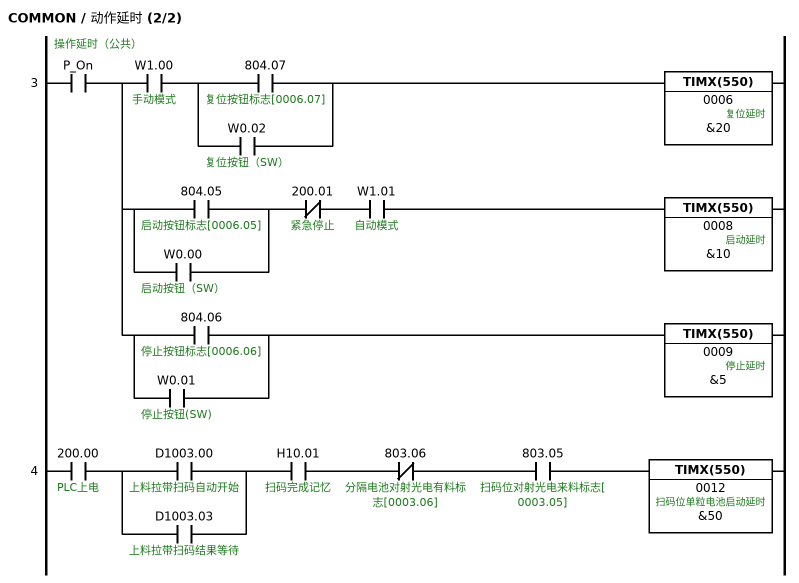
; [picture p168: COMMON / 动作延时, rungs 3-4]
; rung 3: 操作延时（公共）
LD P_On
OUT TR0
AND W1.00  ; 手动模式
LD 804.07  ; 复位按钮标志[0006.07]
OR W0.02  ; 复位按钮（SW）
ANDLD
TIMX(550) 0006 &20  ; 复位延时
LD TR0
LD 804.05  ; 启动按钮标志[0006.05]
OR W0.00  ; 启动按钮（SW）
ANDLD
ANDNOT 200.01  ; 紧急停止
AND W1.01  ; 自动模式
TIMX(550) 0008 &10  ; 启动延时
LD TR0
LD 804.06  ; 停止按钮标志[0006.06]
OR W0.01  ; 停止按钮(SW)
ANDLD
TIMX(550) 0009 &5  ; 停止延时
; rung 4
LD 200.00  ; PLC上电
LD D1003.00  ; 上料拉带扫码自动开始
OR D1003.03  ; 上料拉带扫码结果等待
ANDLD
AND H10.01  ; 扫码完成记忆
ANDNOT 803.06  ; 分隔电池对射光电有料标志[0003.06]
AND 803.05  ; 扫码位对射光电来料标志[0003.05]
TIMX(550) 0012 &50  ; 扫码位单粒电池启动延时

### Section 数据传输

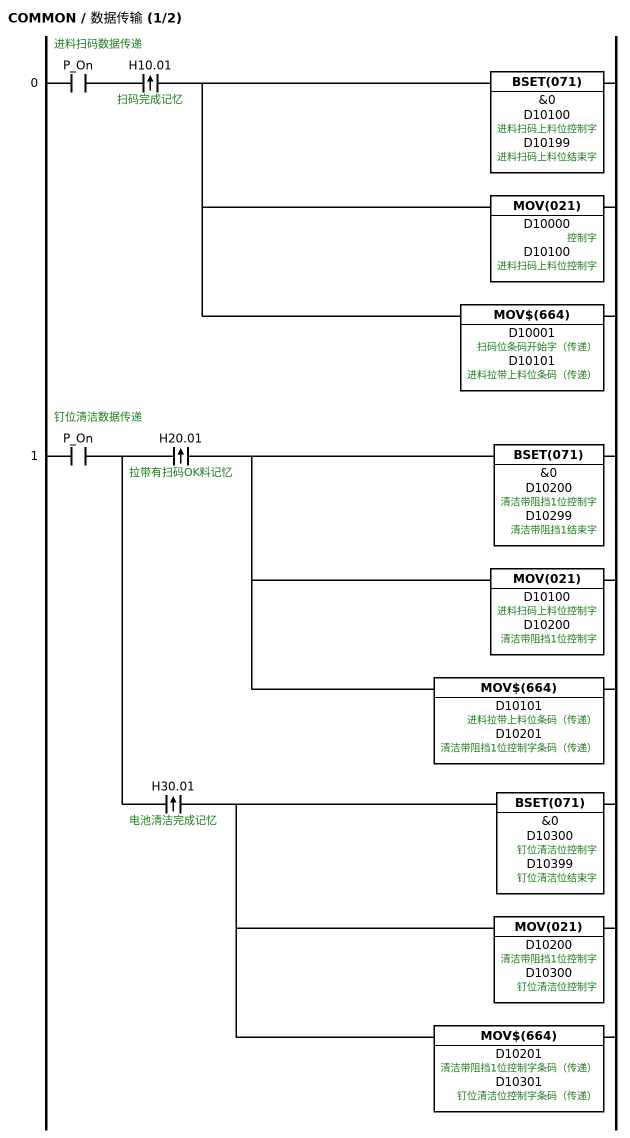
; rung 0: 进料扫码数据传递
LD P_On
@AND H10.01  ; 扫码完成记忆
BSET(071) &0 D10100 D10199  ; 进料扫码上料位控制字, 进料扫码上料位结束字
MOV(021) D10000 D10100  ; 控制字, 进料扫码上料位控制字
MOV$(664) D10001 D10101  ; 扫码位条码开始字（传递）, 进料拉带上料位条码（传递）
; rung 1: 钉位清洁数据传递
LD P_On
OUT TR0
@AND H20.01  ; 拉带有扫码OK料记忆
BSET(071) &0 D10200 D10299  ; 清洁带阻挡1位控制字, 清洁带阻挡1结束字
MOV(021) D10100 D10200  ; 进料扫码上料位控制字, 清洁带阻挡1位控制字
MOV$(664) D10101 D10201  ; 进料拉带上料位条码（传递）, 清洁带阻挡1位控制字条码（传递）
LD TR0
@AND H30.01  ; 电池清洁完成记忆
BSET(071) &0 D10300 D10399  ; 钉位清洁位控制字, 钉位清洁位结束字
MOV(021) D10200 D10300  ; 清洁带阻挡1位控制字, 钉位清洁位控制字
MOV$(664) D10201 D10301  ; 清洁带阻挡1位控制字条码（传递）, 钉位清洁位控制字条码（传递）

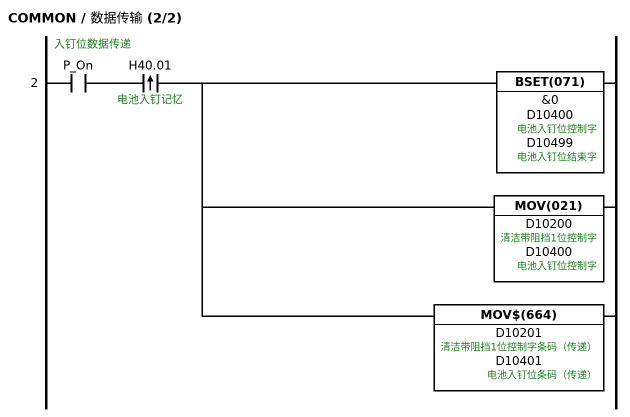
; rung 2: 入钉位数据传递
LD P_On
@AND H40.01  ; 电池入钉记忆
BSET(071) &0 D10400 D10499  ; 电池入钉位控制字, 电池入钉位结束字
MOV(021) D10200 D10400  ; 清洁带阻挡1位控制字, 电池入钉位控制字
MOV$(664) D10201 D10401  ; 清洁带阻挡1位控制字条码（传递）, 电池入钉位条码（传递）

### Section 数据处理

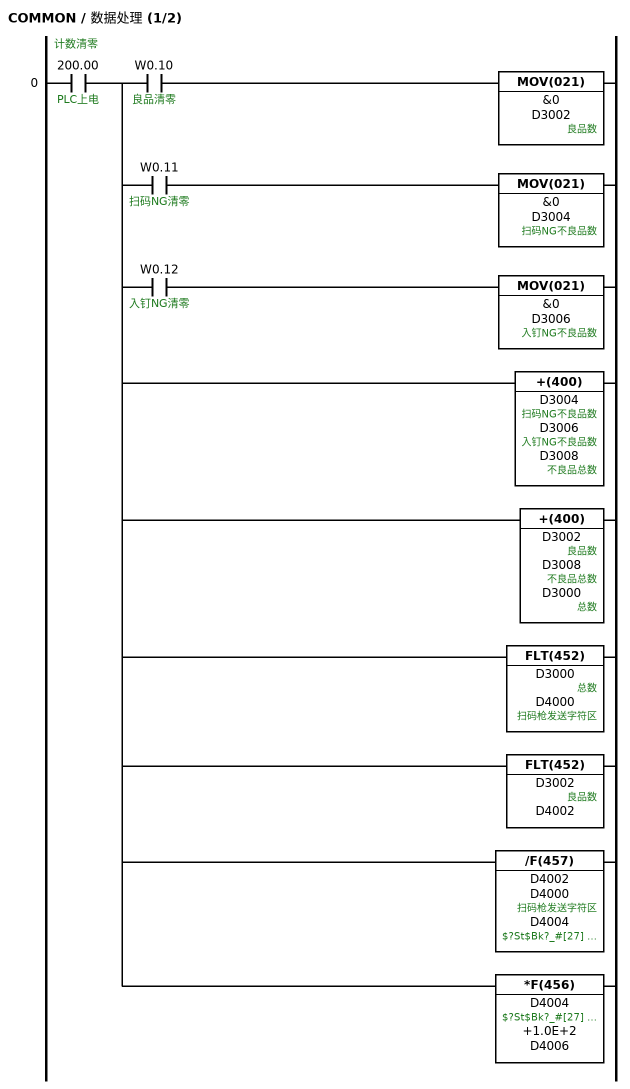
; rung 0: 计数清零
LD 200.00  ; PLC上电
OUT TR0
AND W0.10  ; 良品清零
MOV(021) &0 D3002  ; 良品数
LD TR0
AND W0.11  ; 扫码NG清零
MOV(021) &0 D3004  ; 扫码NG不良品数
LD TR0
AND W0.12  ; 入钉NG清零
MOV(021) &0 D3006  ; 入钉NG不良品数
LD TR0
+(400) D3004 D3006 D3008  ; 扫码NG不良品数, 入钉NG不良品数, 不良品总数
+(400) D3002 D3008 D3000  ; 良品数, 不良品总数, 总数
FLT(452) D3000 D4000  ; 总数, 扫码枪发送字符区
FLT(452) D3002 D4002  ; 良品数
/F(457) D4002 D4000 D4004  ; 扫码枪发送字符区, $?St$Bk?_#[27] / "OK"$?St$Bk?_#[27]
*F(456) D4004 +1.0E+2 D4006  ; $?St$Bk?_#[27] / "OK"$?St$Bk?_#[27]

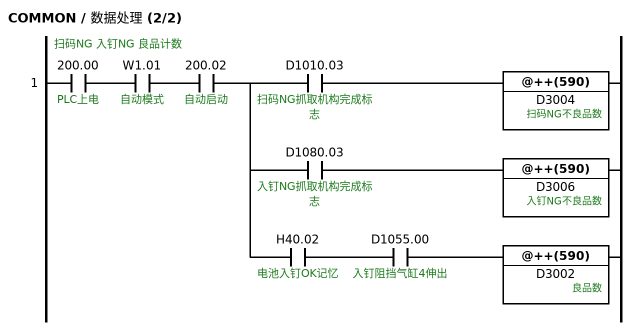
; rung 1: 扫码NG 入钉NG 良品计数
LD 200.00  ; PLC上电
AND W1.01  ; 自动模式
AND 200.02  ; 自动启动
OUT TR0
AND D1010.03  ; 扫码NG抓取机构完成标志
@++(590) D3004  ; 扫码NG不良品数
LD TR0
AND D1080.03  ; 入钉NG抓取机构完成标志
@++(590) D3006  ; 入钉NG不良品数
LD TR0
AND H40.02  ; 电池入钉OK记忆
AND D1055.00  ; 入钉阻挡气缸4伸出
@++(590) D3002  ; 良品数

### Section 报警程序

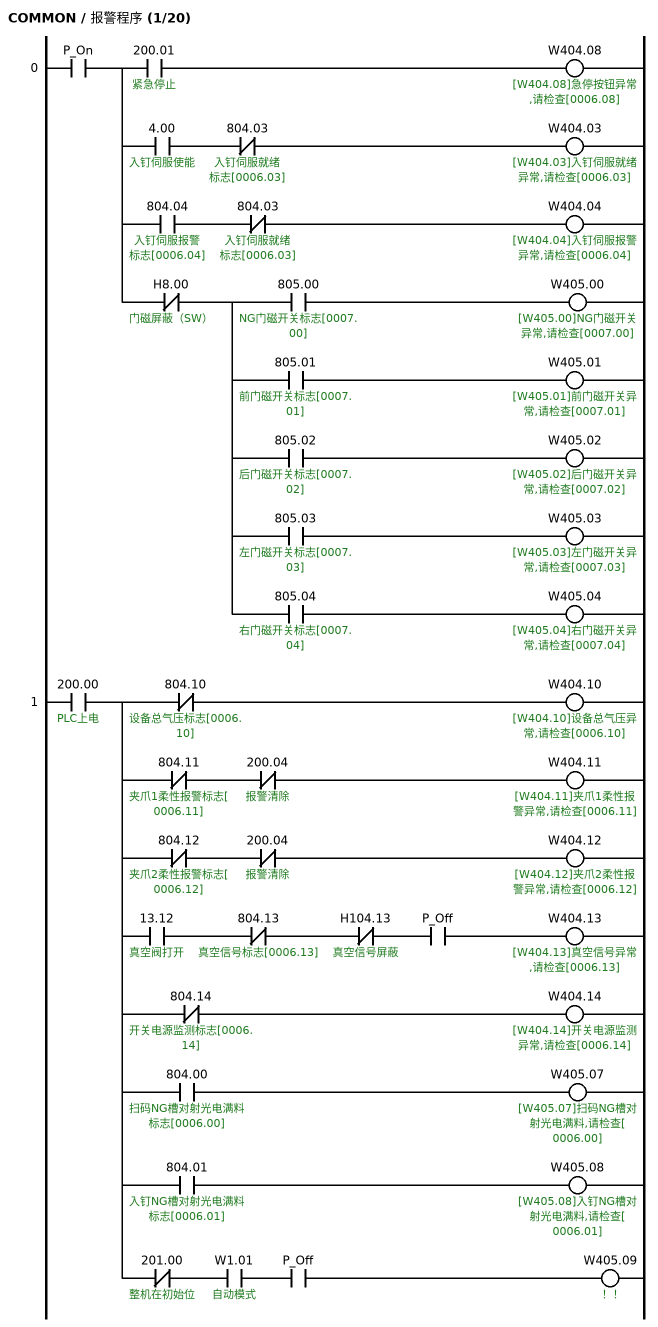
; rung 0
LD P_On
OUT TR0
AND 200.01  ; 紧急停止
OUT W404.08  ; [W404.08]急停按钮异常,请检查[0006.08]
LD TR0
AND 4.00  ; 入钉伺服使能
ANDNOT 804.03  ; 入钉伺服就绪 标志[0006.03]
OUT W404.03  ; [W404.03]入钉伺服就绪异常,请检查[0006.03]
LD TR0
AND 804.04  ; 入钉伺服报警 标志[0006.04]
ANDNOT 804.03  ; 入钉伺服就绪 标志[0006.03]
OUT W404.04  ; [W404.04]入钉伺服报警异常,请检查[0006.04]
LD TR0
ANDNOT H8.00  ; 门磁屏蔽（SW）
OUT TR0
AND 805.00  ; NG门磁开关标志[0007.00]
OUT W405.00  ; [W405.00]NG门磁开关异常,请检查[0007.00]
LD TR0
AND 805.01  ; 前门磁开关标志[0007.01]
OUT W405.01  ; [W405.01]前门磁开关异常,请检查[0007.01]
LD TR0
AND 805.02  ; 后门磁开关标志[0007.02]
OUT W405.02  ; [W405.02]后门磁开关异常,请检查[0007.02]
LD TR0
AND 805.03  ; 左门磁开关标志[0007.03]
OUT W405.03  ; [W405.03]左门磁开关异常,请检查[0007.03]
LD TR0
AND 805.04  ; 右门磁开关标志[0007.04]
OUT W405.04  ; [W405.04]右门磁开关异常,请检查[0007.04]
; rung 1
LD 200.00  ; PLC上电
OUT TR0
ANDNOT 804.10  ; 设备总气压标志[0006.10]
OUT W404.10  ; [W404.10]设备总气压异常,请检查[0006.10]
LD TR0
ANDNOT 804.11  ; 夹爪1柔性报警标志[0006.11]
ANDNOT 200.04  ; 报警清除
OUT W404.11  ; [W404.11]夹爪1柔性报警异常,请检查[0006.11]
LD TR0
ANDNOT 804.12  ; 夹爪2柔性报警标志[0006.12]
ANDNOT 200.04  ; 报警清除
OUT W404.12  ; [W404.12]夹爪2柔性报警异常,请检查[0006.12]
LD TR0
AND 13.12  ; 真空阀打开
ANDNOT 804.13  ; 真空信号标志[0006.13]
ANDNOT H104.13  ; 真空信号屏蔽
AND P_Off
OUT W404.13  ; [W404.13]真空信号异常,请检查[0006.13]
LD TR0
ANDNOT 804.14  ; 开关电源监测标志[0006.14]
OUT W404.14  ; [W404.14]开关电源监测异常,请检查[0006.14]
LD TR0
AND 804.00  ; 扫码NG槽对射光电满料标志[0006.00]
OUT W405.07  ; [W405.07]扫码NG槽对射光电满料,请检查[0006.00]
LD TR0
AND 804.01  ; 入钉NG槽对射光电满料标志[0006.01]
OUT W405.08  ; [W405.08]入钉NG槽对射光电满料,请检查[0006.01]
LD TR0
ANDNOT 201.00  ; 整机在初始位
AND W1.01  ; 自动模式
AND P_Off
OUT W405.09  ; ！！

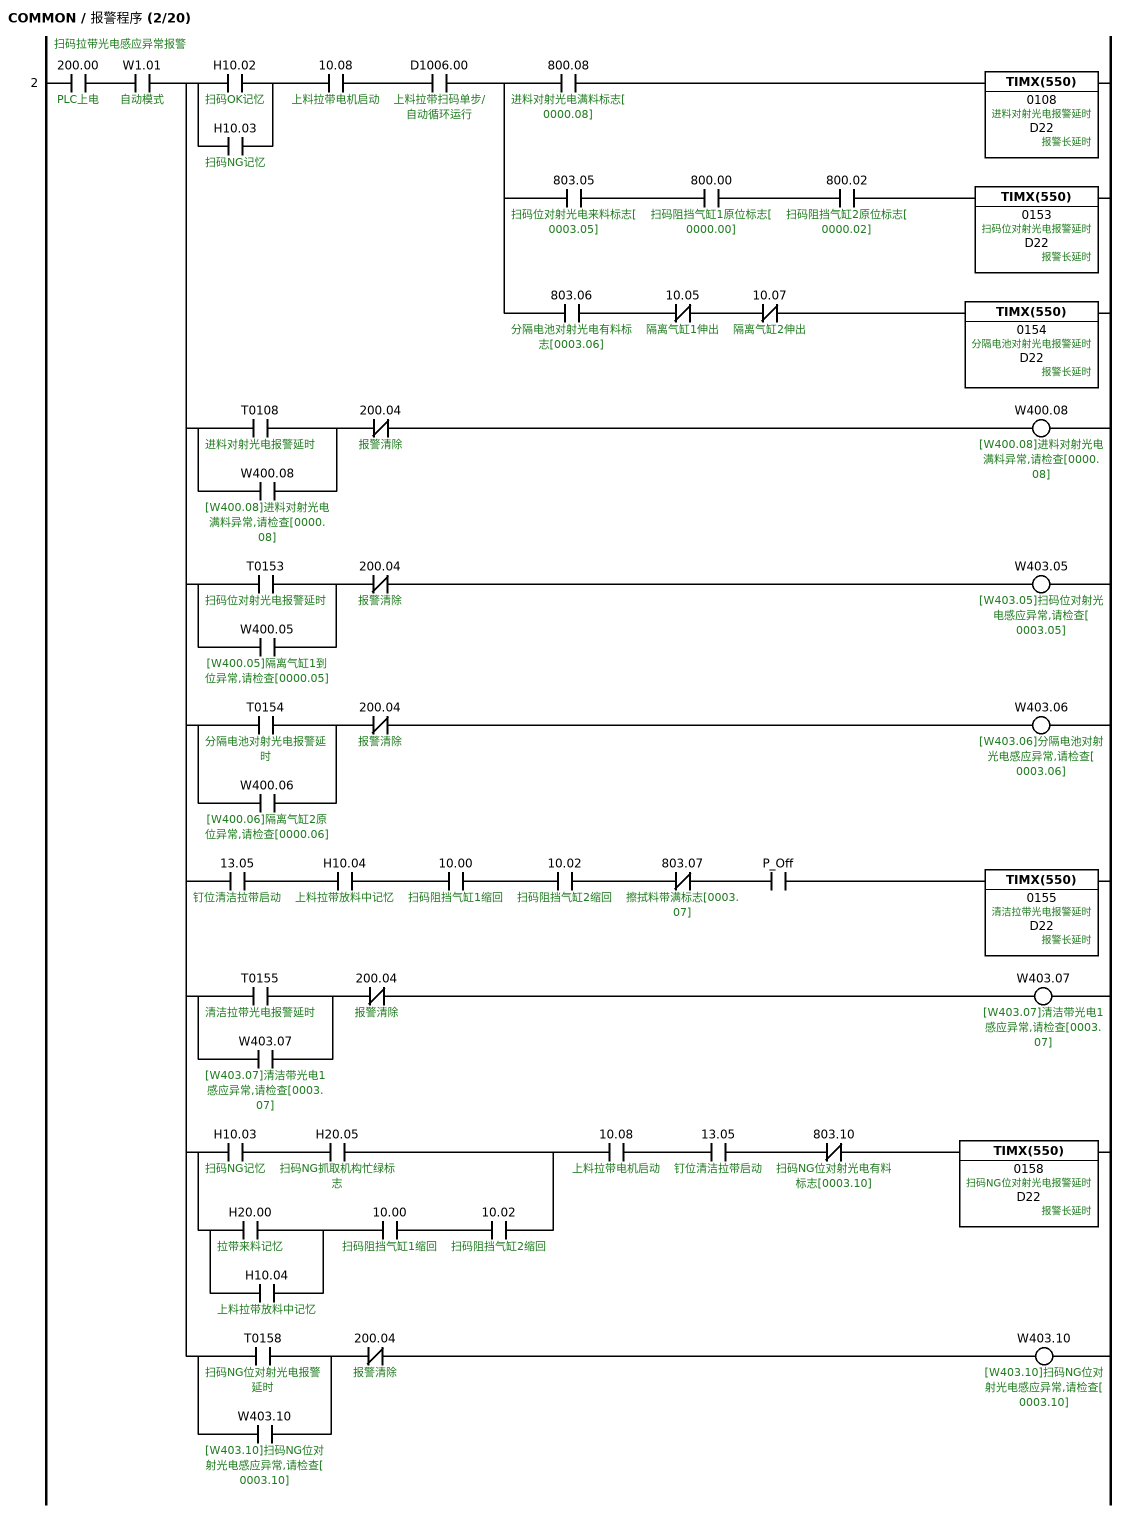
; rung 2: 扫码拉带光电感应异常报警
LD 200.00  ; PLC上电
AND W1.01  ; 自动模式
OUT TR0
LD H10.02  ; 扫码OK记忆
OR H10.03  ; 扫码NG记忆
ANDLD
AND 10.08  ; 上料拉带电机启动
AND D1006.00  ; 上料拉带扫码单步/自动循环运行
OUT TR1
AND 800.08  ; 进料对射光电满料标志[0000.08]
TIMX(550) 0108 D22  ; 报警长延时, 进料对射光电报警延时
LD TR1
AND 803.05  ; 扫码位对射光电来料标志[0003.05]
AND 800.00  ; 扫码阻挡气缸1原位标志[0000.00]
AND 800.02  ; 扫码阻挡气缸2原位标志[0000.02]
TIMX(550) 0153 D22  ; 报警长延时, 扫码位对射光电报警延时
LD TR1
AND 803.06  ; 分隔电池对射光电有料标志[0003.06]
ANDNOT 10.05  ; 隔离气缸1伸出
ANDNOT 10.07  ; 隔离气缸2伸出
TIMX(550) 0154 D22  ; 报警长延时, 分隔电池对射光电报警延时
LD TR0
LD T0108  ; 进料对射光电报警延时
OR W400.08  ; [W400.08]进料对射光电满料异常,请检查[0000.08]
ANDLD
ANDNOT 200.04  ; 报警清除
OUT W400.08  ; [W400.08]进料对射光电满料异常,请检查[0000.08]
LD TR0
LD T0153  ; 扫码位对射光电报警延时
OR W400.05  ; [W400.05]隔离气缸1到位异常,请检查[0000.05]
ANDLD
ANDNOT 200.04  ; 报警清除
OUT W403.05  ; [W403.05]扫码位对射光电感应异常,请检查[0003.05]
LD TR0
LD T0154  ; 分隔电池对射光电报警延时
OR W400.06  ; [W400.06]隔离气缸2原位异常,请检查[0000.06]
ANDLD
ANDNOT 200.04  ; 报警清除
OUT W403.06  ; [W403.06]分隔电池对射光电感应异常,请检查[0003.06]
LD TR0
AND 13.05  ; 钉位清洁拉带启动
AND H10.04  ; 上料拉带放料中记忆
AND 10.00  ; 扫码阻挡气缸1缩回
AND 10.02  ; 扫码阻挡气缸2缩回
ANDNOT 803.07  ; 擦拭料带满标志[0003.07]
AND P_Off
TIMX(550) 0155 D22  ; 报警长延时, 清洁拉带光电报警延时
LD TR0
LD T0155  ; 清洁拉带光电报警延时
OR W403.07  ; [W403.07]清洁带光电1感应异常,请检查[0003.07]
ANDLD
ANDNOT 200.04  ; 报警清除
OUT W403.07  ; [W403.07]清洁带光电1感应异常,请检查[0003.07]
LD TR0
LD H10.03  ; 扫码NG记忆
AND H20.05  ; 扫码NG抓取机构忙绿标志
LD H20.00  ; 拉带来料记忆
OR H10.04  ; 上料拉带放料中记忆
AND 10.00  ; 扫码阻挡气缸1缩回
AND 10.02  ; 扫码阻挡气缸2缩回
ORLD
ANDLD
AND 10.08  ; 上料拉带电机启动
AND 13.05  ; 钉位清洁拉带启动
ANDNOT 803.10  ; 扫码NG位对射光电有料标志[0003.10]
TIMX(550) 0158 D22  ; 报警长延时, 扫码NG位对射光电报警延时
LD TR0
LD T0158  ; 扫码NG位对射光电报警延时
OR W403.10  ; [W403.10]扫码NG位对射光电感应异常,请检查[0003.10]
ANDLD
ANDNOT 200.04  ; 报警清除
OUT W403.10  ; [W403.10]扫码NG位对射光电感应异常,请检查[0003.10]

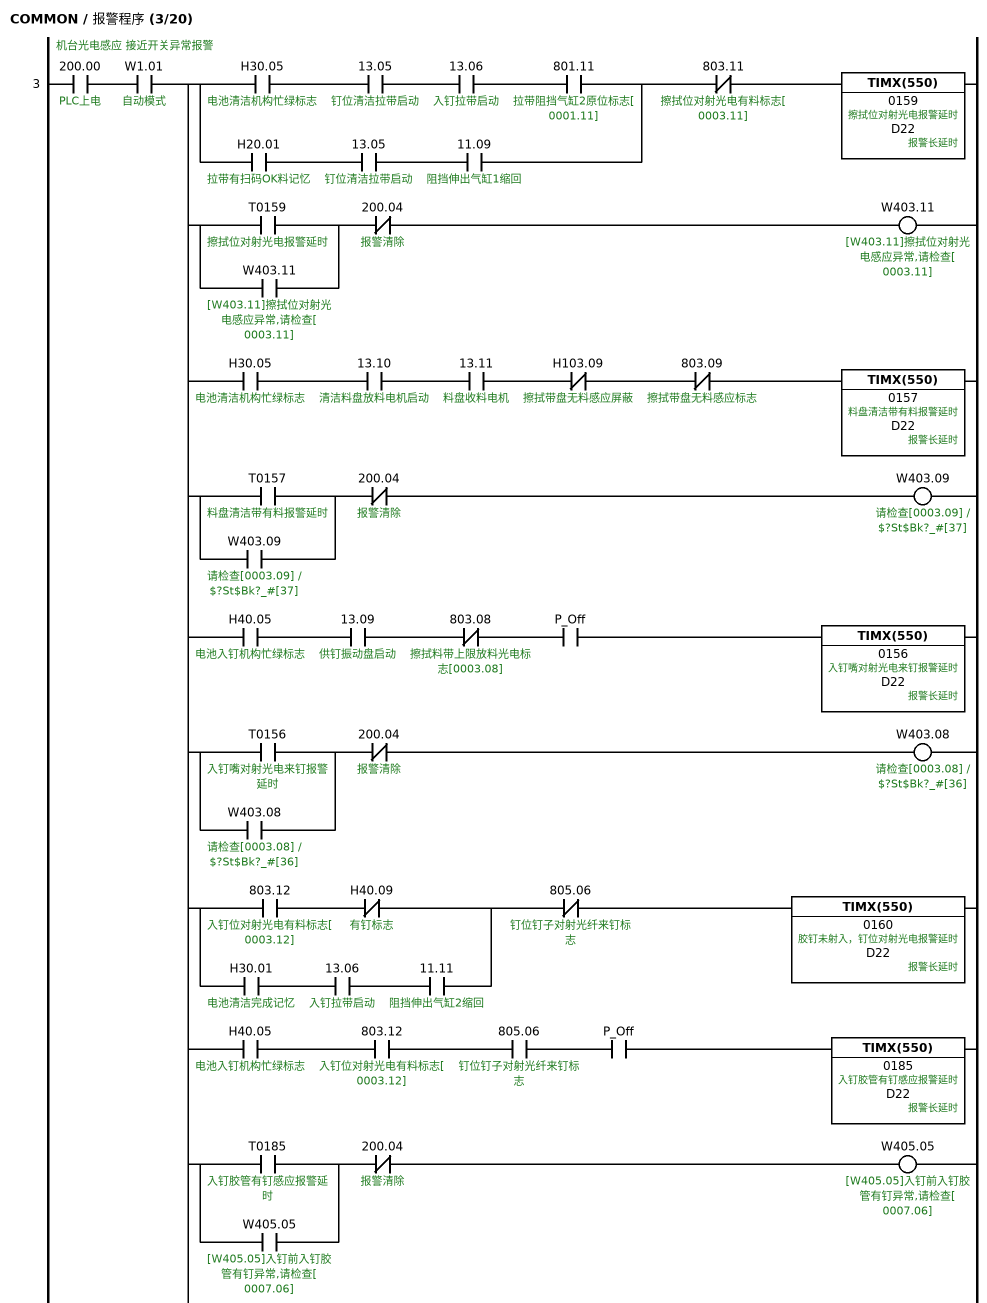

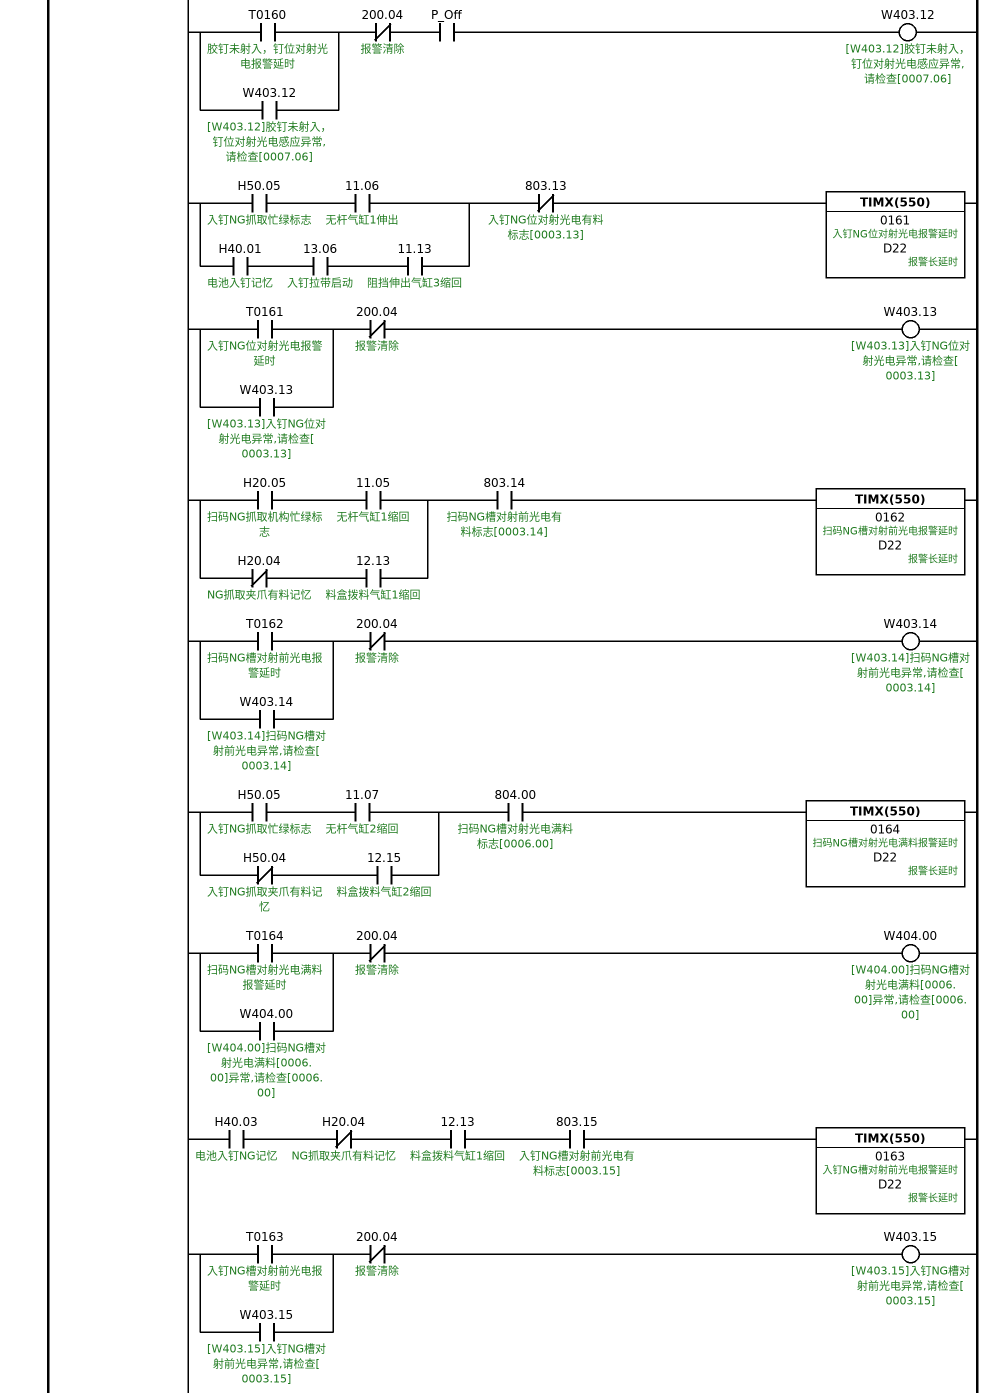

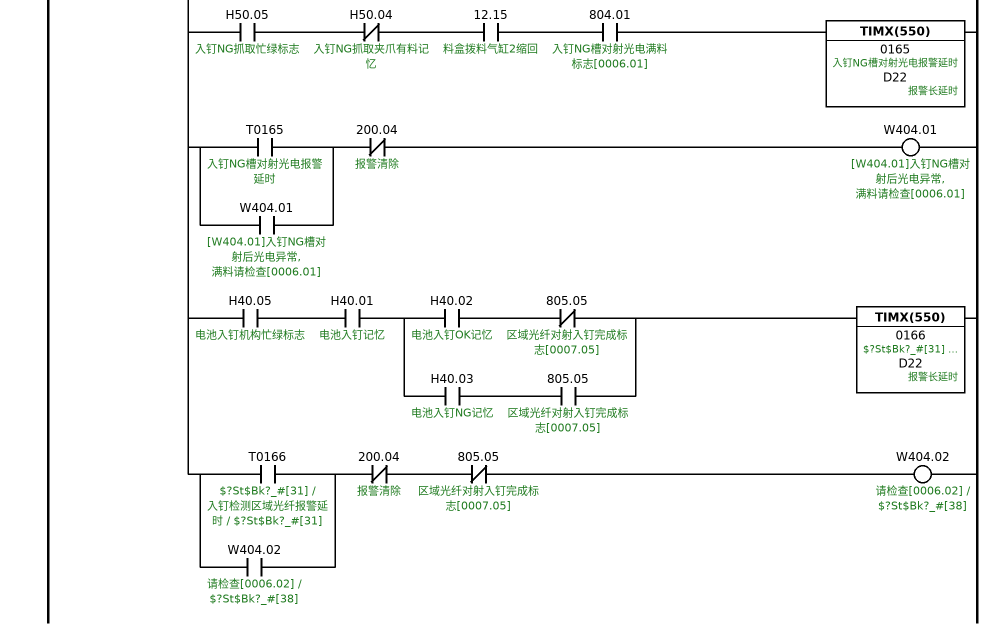
; rung 3: 机台光电感应 接近开关异常报警
LD 200.00  ; PLC上电
AND W1.01  ; 自动模式
OUT TR0
LD H30.05  ; 电池清洁机构忙绿标志
AND 13.05  ; 钉位清洁拉带启动
AND 13.06  ; 入钉拉带启动
AND 801.11  ; 拉带阻挡气缸2原位标志[0001.11]
LD H20.01  ; 拉带有扫码OK料记忆
AND 13.05  ; 钉位清洁拉带启动
AND 11.09  ; 阻挡伸出气缸1缩回
ORLD
ANDLD
ANDNOT 803.11  ; 擦拭位对射光电有料标志[0003.11]
TIMX(550) 0159 D22  ; 报警长延时, 擦拭位对射光电报警延时
LD TR0
LD T0159  ; 擦拭位对射光电报警延时
OR W403.11  ; [W403.11]擦拭位对射光电感应异常,请检查[0003.11]
ANDLD
ANDNOT 200.04  ; 报警清除
OUT W403.11  ; [W403.11]擦拭位对射光电感应异常,请检查[0003.11]
LD TR0
AND H30.05  ; 电池清洁机构忙绿标志
AND 13.10  ; 清洁料盘放料电机启动
AND 13.11  ; 料盘收料电机
ANDNOT H103.09  ; 擦拭带盘无料感应屏蔽
ANDNOT 803.09  ; 擦拭带盘无料感应标志
TIMX(550) 0157 D22  ; 报警长延时, 料盘清洁带有料报警延时
LD TR0
LD T0157  ; 料盘清洁带有料报警延时
OR W403.09  ; 请检查[0003.09] / $?St$Bk?_#[37]
ANDLD
ANDNOT 200.04  ; 报警清除
OUT W403.09  ; 请检查[0003.09] / $?St$Bk?_#[37]
LD TR0
AND H40.05  ; 电池入钉机构忙绿标志
AND 13.09  ; 供钉振动盘启动
ANDNOT 803.08  ; 擦拭料带上限放料光电标志[0003.08]
AND P_Off
TIMX(550) 0156 D22  ; 报警长延时, 入钉嘴对射光电来钉报警延时
LD TR0
LD T0156  ; 入钉嘴对射光电来钉报警延时
OR W403.08  ; 请检查[0003.08] / $?St$Bk?_#[36]
ANDLD
ANDNOT 200.04  ; 报警清除
OUT W403.08  ; 请检查[0003.08] / $?St$Bk?_#[36]
LD TR0
LD 803.12  ; 入钉位对射光电有料标志[0003.12]
ANDNOT H40.09  ; 有钉标志
LD H30.01  ; 电池清洁完成记忆
AND 13.06  ; 入钉拉带启动
AND 11.11  ; 阻挡伸出气缸2缩回
ORLD
ANDLD
ANDNOT 805.06  ; 钉位钉子对射光纤来钉标志
TIMX(550) 0160 D22  ; 报警长延时, 胶钉未射入，钉位对射光电报警延时
LD TR0
AND H40.05  ; 电池入钉机构忙绿标志
AND 803.12  ; 入钉位对射光电有料标志[0003.12]
AND 805.06  ; 钉位钉子对射光纤来钉标志
AND P_Off
TIMX(550) 0185 D22  ; 报警长延时, 入钉胶管有钉感应报警延时
LD TR0
LD T0185  ; 入钉胶管有钉感应报警延时
OR W405.05  ; [W405.05]入钉前入钉胶管有钉异常,请检查[0007.06]
ANDLD
ANDNOT 200.04  ; 报警清除
OUT W405.05  ; [W405.05]入钉前入钉胶管有钉异常,请检查[0007.06]
LD TR0
LD T0160  ; 胶钉未射入，钉位对射光电报警延时
OR W403.12  ; [W403.12]胶钉未射入，钉位对射光电感应异常,请检查[0007.06]
ANDLD
ANDNOT 200.04  ; 报警清除
AND P_Off
OUT W403.12  ; [W403.12]胶钉未射入，钉位对射光电感应异常,请检查[0007.06]
LD TR0
LD H50.05  ; 入钉NG抓取忙绿标志
AND 11.06  ; 无杆气缸1伸出
LD H40.01  ; 电池入钉记忆
AND 13.06  ; 入钉拉带启动
AND 11.13  ; 阻挡伸出气缸3缩回
ORLD
ANDLD
ANDNOT 803.13  ; 入钉NG位对射光电有料标志[0003.13]
TIMX(550) 0161 D22  ; 报警长延时, 入钉NG位对射光电报警延时
LD TR0
LD T0161  ; 入钉NG位对射光电报警延时
OR W403.13  ; [W403.13]入钉NG位对射光电异常,请检查[0003.13]
ANDLD
ANDNOT 200.04  ; 报警清除
OUT W403.13  ; [W403.13]入钉NG位对射光电异常,请检查[0003.13]
LD TR0
LD H20.05  ; 扫码NG抓取机构忙绿标志
AND 11.05  ; 无杆气缸1缩回
LDNOT H20.04  ; NG抓取夹爪有料记忆
AND 12.13  ; 料盒拨料气缸1缩回
ORLD
ANDLD
AND 803.14  ; 扫码NG槽对射前光电有料标志[0003.14]
TIMX(550) 0162 D22  ; 报警长延时, 扫码NG槽对射前光电报警延时
LD TR0
LD T0162  ; 扫码NG槽对射前光电报警延时
OR W403.14  ; [W403.14]扫码NG槽对射前光电异常,请检查[0003.14]
ANDLD
ANDNOT 200.04  ; 报警清除
OUT W403.14  ; [W403.14]扫码NG槽对射前光电异常,请检查[0003.14]
LD TR0
LD H50.05  ; 入钉NG抓取忙绿标志
AND 11.07  ; 无杆气缸2缩回
LDNOT H50.04  ; 入钉NG抓取夹爪有料记忆
AND 12.15  ; 料盒拨料气缸2缩回
ORLD
ANDLD
AND 804.00  ; 扫码NG槽对射光电满料标志[0006.00]
TIMX(550) 0164 D22  ; 报警长延时, 扫码NG槽对射光电满料报警延时
LD TR0
LD T0164  ; 扫码NG槽对射光电满料报警延时
OR W404.00  ; [W404.00]扫码NG槽对射光电满料[0006.00]异常,请检查[0006.00]
ANDLD
ANDNOT 200.04  ; 报警清除
OUT W404.00  ; [W404.00]扫码NG槽对射光电满料[0006.00]异常,请检查[0006.00]
LD TR0
AND H40.03  ; 电池入钉NG记忆
ANDNOT H20.04  ; NG抓取夹爪有料记忆
AND 12.13  ; 料盒拨料气缸1缩回
AND 803.15  ; 入钉NG槽对射前光电有料标志[0003.15]
TIMX(550) 0163 D22  ; 报警长延时, 入钉NG槽对射前光电报警延时
LD TR0
LD T0163  ; 入钉NG槽对射前光电报警延时
OR W403.15  ; [W403.15]入钉NG槽对射前光电异常,请检查[0003.15]
ANDLD
ANDNOT 200.04  ; 报警清除
OUT W403.15  ; [W403.15]入钉NG槽对射前光电异常,请检查[0003.15]
LD TR0
AND H50.05  ; 入钉NG抓取忙绿标志
ANDNOT H50.04  ; 入钉NG抓取夹爪有料记忆
AND 12.15  ; 料盒拨料气缸2缩回
AND 804.01  ; 入钉NG槽对射光电满料标志[0006.01]
TIMX(550) 0165 D22  ; 报警长延时, 入钉NG槽对射光电报警延时
LD TR0
LD T0165  ; 入钉NG槽对射光电报警延时
OR W404.01  ; [W404.01]入钉NG槽对射后光电异常,满料请检查[0006.01]
ANDLD
ANDNOT 200.04  ; 报警清除
OUT W404.01  ; [W404.01]入钉NG槽对射后光电异常,满料请检查[0006.01]
LD TR0
AND H40.05  ; 电池入钉机构忙绿标志
AND H40.01  ; 电池入钉记忆
LD H40.02  ; 电池入钉OK记忆
ANDNOT 805.05  ; 区域光纤对射入钉完成标志[0007.05]
LD H40.03  ; 电池入钉NG记忆
AND 805.05  ; 区域光纤对射入钉完成标志[0007.05]
ORLD
ANDLD
TIMX(550) 0166 D22  ; 报警长延时, $?St$Bk?_#[31] / 入钉检测区域光纤报警延时 / $?St$Bk?_#[31]
LD TR0
LD T0166  ; $?St$Bk?_#[31] / 入钉检测区域光纤报警延时 / $?St$Bk?_#[31]
OR W404.02  ; 请检查[0006.02] / $?St$Bk?_#[38]
ANDLD
ANDNOT 200.04  ; 报警清除
ANDNOT 805.05  ; 区域光纤对射入钉完成标志[0007.05]
OUT W404.02  ; 请检查[0006.02] / $?St$Bk?_#[38]

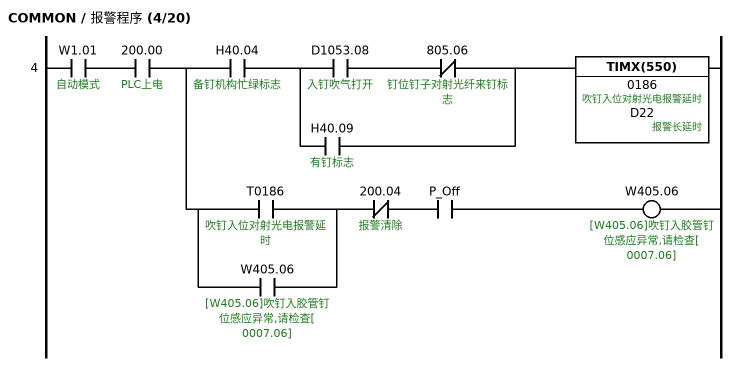
; rung 4
LD W1.01  ; 自动模式
AND 200.00  ; PLC上电
OUT TR0
AND H40.04  ; 备钉机构忙绿标志
LD D1053.08  ; 入钉吹气打开
ANDNOT 805.06  ; 钉位钉子对射光纤来钉标志
OR H40.09  ; 有钉标志
ANDLD
TIMX(550) 0186 D22  ; 报警长延时, 吹钉入位对射光电报警延时
LD TR0
LD T0186  ; 吹钉入位对射光电报警延时
OR W405.06  ; [W405.06]吹钉入胶管钉位感应异常,请检查[0007.06]
ANDLD
ANDNOT 200.04  ; 报警清除
AND P_Off
OUT W405.06  ; [W405.06]吹钉入胶管钉位感应异常,请检查[0007.06]

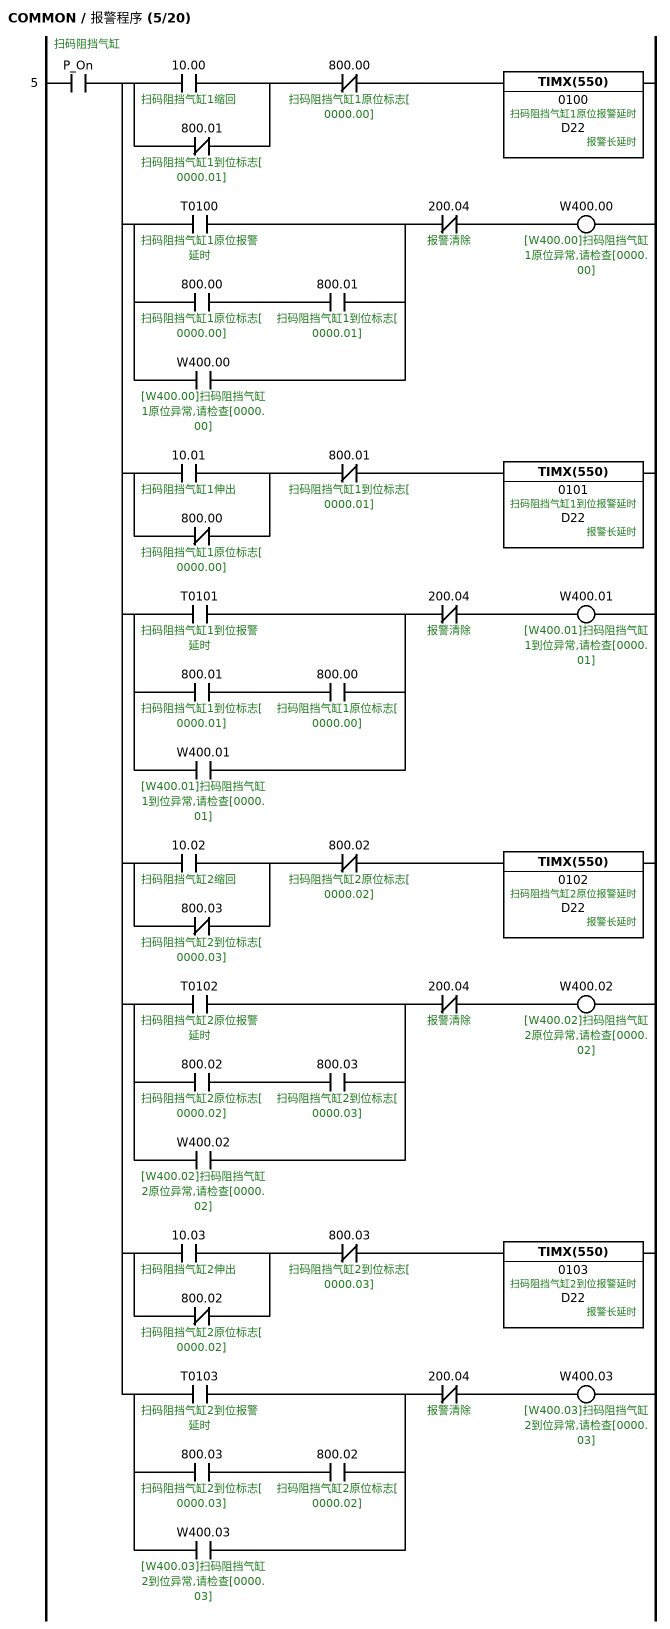
; rung 5: 扫码阻挡气缸
LD P_On
OUT TR0
LD 10.00  ; 扫码阻挡气缸1缩回
ORNOT 800.01  ; 扫码阻挡气缸1到位标志[0000.01]
ANDLD
ANDNOT 800.00  ; 扫码阻挡气缸1原位标志[0000.00]
TIMX(550) 0100 D22  ; 报警长延时, 扫码阻挡气缸1原位报警延时
LD TR0
LD T0100  ; 扫码阻挡气缸1原位报警延时
LD 800.00  ; 扫码阻挡气缸1原位标志[0000.00]
AND 800.01  ; 扫码阻挡气缸1到位标志[0000.01]
ORLD
OR W400.00  ; [W400.00]扫码阻挡气缸1原位异常,请检查[0000.00]
ANDLD
ANDNOT 200.04  ; 报警清除
OUT W400.00  ; [W400.00]扫码阻挡气缸1原位异常,请检查[0000.00]
LD TR0
LD 10.01  ; 扫码阻挡气缸1伸出
ORNOT 800.00  ; 扫码阻挡气缸1原位标志[0000.00]
ANDLD
ANDNOT 800.01  ; 扫码阻挡气缸1到位标志[0000.01]
TIMX(550) 0101 D22  ; 报警长延时, 扫码阻挡气缸1到位报警延时
LD TR0
LD T0101  ; 扫码阻挡气缸1到位报警延时
LD 800.01  ; 扫码阻挡气缸1到位标志[0000.01]
AND 800.00  ; 扫码阻挡气缸1原位标志[0000.00]
ORLD
OR W400.01  ; [W400.01]扫码阻挡气缸1到位异常,请检查[0000.01]
ANDLD
ANDNOT 200.04  ; 报警清除
OUT W400.01  ; [W400.01]扫码阻挡气缸1到位异常,请检查[0000.01]
LD TR0
LD 10.02  ; 扫码阻挡气缸2缩回
ORNOT 800.03  ; 扫码阻挡气缸2到位标志[0000.03]
ANDLD
ANDNOT 800.02  ; 扫码阻挡气缸2原位标志[0000.02]
TIMX(550) 0102 D22  ; 报警长延时, 扫码阻挡气缸2原位报警延时
LD TR0
LD T0102  ; 扫码阻挡气缸2原位报警延时
LD 800.02  ; 扫码阻挡气缸2原位标志[0000.02]
AND 800.03  ; 扫码阻挡气缸2到位标志[0000.03]
ORLD
OR W400.02  ; [W400.02]扫码阻挡气缸2原位异常,请检查[0000.02]
ANDLD
ANDNOT 200.04  ; 报警清除
OUT W400.02  ; [W400.02]扫码阻挡气缸2原位异常,请检查[0000.02]
LD TR0
LD 10.03  ; 扫码阻挡气缸2伸出
ORNOT 800.02  ; 扫码阻挡气缸2原位标志[0000.02]
ANDLD
ANDNOT 800.03  ; 扫码阻挡气缸2到位标志[0000.03]
TIMX(550) 0103 D22  ; 报警长延时, 扫码阻挡气缸2到位报警延时
LD TR0
LD T0103  ; 扫码阻挡气缸2到位报警延时
LD 800.03  ; 扫码阻挡气缸2到位标志[0000.03]
AND 800.02  ; 扫码阻挡气缸2原位标志[0000.02]
ORLD
OR W400.03  ; [W400.03]扫码阻挡气缸2到位异常,请检查[0000.03]
ANDLD
ANDNOT 200.04  ; 报警清除
OUT W400.03  ; [W400.03]扫码阻挡气缸2到位异常,请检查[0000.03]

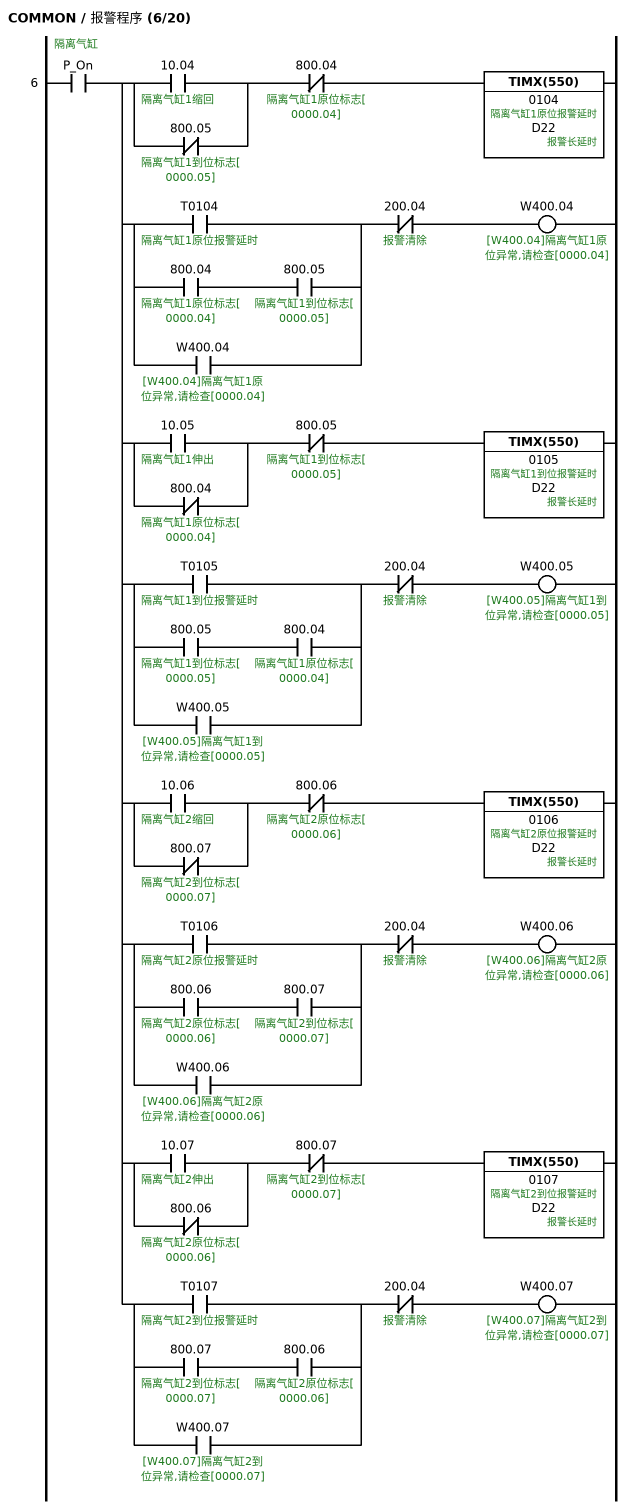
; rung 6: 隔离气缸
LD P_On
OUT TR0
LD 10.04  ; 隔离气缸1缩回
ORNOT 800.05  ; 隔离气缸1到位标志[0000.05]
ANDLD
ANDNOT 800.04  ; 隔离气缸1原位标志[0000.04]
TIMX(550) 0104 D22  ; 报警长延时, 隔离气缸1原位报警延时
LD TR0
LD T0104  ; 隔离气缸1原位报警延时
LD 800.04  ; 隔离气缸1原位标志[0000.04]
AND 800.05  ; 隔离气缸1到位标志[0000.05]
ORLD
OR W400.04  ; [W400.04]隔离气缸1原位异常,请检查[0000.04]
ANDLD
ANDNOT 200.04  ; 报警清除
OUT W400.04  ; [W400.04]隔离气缸1原位异常,请检查[0000.04]
LD TR0
LD 10.05  ; 隔离气缸1伸出
ORNOT 800.04  ; 隔离气缸1原位标志[0000.04]
ANDLD
ANDNOT 800.05  ; 隔离气缸1到位标志[0000.05]
TIMX(550) 0105 D22  ; 报警长延时, 隔离气缸1到位报警延时
LD TR0
LD T0105  ; 隔离气缸1到位报警延时
LD 800.05  ; 隔离气缸1到位标志[0000.05]
AND 800.04  ; 隔离气缸1原位标志[0000.04]
ORLD
OR W400.05  ; [W400.05]隔离气缸1到位异常,请检查[0000.05]
ANDLD
ANDNOT 200.04  ; 报警清除
OUT W400.05  ; [W400.05]隔离气缸1到位异常,请检查[0000.05]
LD TR0
LD 10.06  ; 隔离气缸2缩回
ORNOT 800.07  ; 隔离气缸2到位标志[0000.07]
ANDLD
ANDNOT 800.06  ; 隔离气缸2原位标志[0000.06]
TIMX(550) 0106 D22  ; 报警长延时, 隔离气缸2原位报警延时
LD TR0
LD T0106  ; 隔离气缸2原位报警延时
LD 800.06  ; 隔离气缸2原位标志[0000.06]
AND 800.07  ; 隔离气缸2到位标志[0000.07]
ORLD
OR W400.06  ; [W400.06]隔离气缸2原位异常,请检查[0000.06]
ANDLD
ANDNOT 200.04  ; 报警清除
OUT W400.06  ; [W400.06]隔离气缸2原位异常,请检查[0000.06]
LD TR0
LD 10.07  ; 隔离气缸2伸出
ORNOT 800.06  ; 隔离气缸2原位标志[0000.06]
ANDLD
ANDNOT 800.07  ; 隔离气缸2到位标志[0000.07]
TIMX(550) 0107 D22  ; 报警长延时, 隔离气缸2到位报警延时
LD TR0
LD T0107  ; 隔离气缸2到位报警延时
LD 800.07  ; 隔离气缸2到位标志[0000.07]
AND 800.06  ; 隔离气缸2原位标志[0000.06]
ORLD
OR W400.07  ; [W400.07]隔离气缸2到位异常,请检查[0000.07]
ANDLD
ANDNOT 200.04  ; 报警清除
OUT W400.07  ; [W400.07]隔离气缸2到位异常,请检查[0000.07]

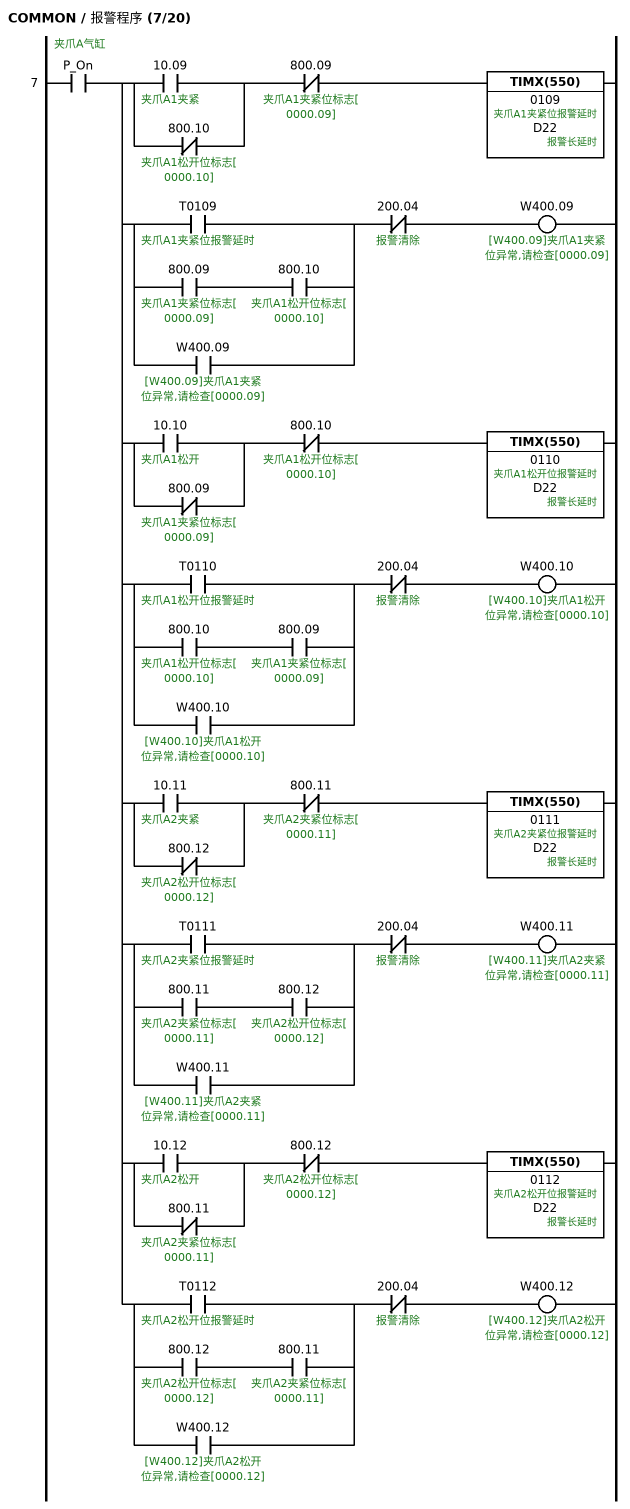
; rung 7: 夹爪A气缸
LD P_On
OUT TR0
LD 10.09  ; 夹爪A1夹紧
ORNOT 800.10  ; 夹爪A1松开位标志[0000.10]
ANDLD
ANDNOT 800.09  ; 夹爪A1夹紧位标志[0000.09]
TIMX(550) 0109 D22  ; 报警长延时, 夹爪A1夹紧位报警延时
LD TR0
LD T0109  ; 夹爪A1夹紧位报警延时
LD 800.09  ; 夹爪A1夹紧位标志[0000.09]
AND 800.10  ; 夹爪A1松开位标志[0000.10]
ORLD
OR W400.09  ; [W400.09]夹爪A1夹紧位异常,请检查[0000.09]
ANDLD
ANDNOT 200.04  ; 报警清除
OUT W400.09  ; [W400.09]夹爪A1夹紧位异常,请检查[0000.09]
LD TR0
LD 10.10  ; 夹爪A1松开
ORNOT 800.09  ; 夹爪A1夹紧位标志[0000.09]
ANDLD
ANDNOT 800.10  ; 夹爪A1松开位标志[0000.10]
TIMX(550) 0110 D22  ; 报警长延时, 夹爪A1松开位报警延时
LD TR0
LD T0110  ; 夹爪A1松开位报警延时
LD 800.10  ; 夹爪A1松开位标志[0000.10]
AND 800.09  ; 夹爪A1夹紧位标志[0000.09]
ORLD
OR W400.10  ; [W400.10]夹爪A1松开位异常,请检查[0000.10]
ANDLD
ANDNOT 200.04  ; 报警清除
OUT W400.10  ; [W400.10]夹爪A1松开位异常,请检查[0000.10]
LD TR0
LD 10.11  ; 夹爪A2夹紧
ORNOT 800.12  ; 夹爪A2松开位标志[0000.12]
ANDLD
ANDNOT 800.11  ; 夹爪A2夹紧位标志[0000.11]
TIMX(550) 0111 D22  ; 报警长延时, 夹爪A2夹紧位报警延时
LD TR0
LD T0111  ; 夹爪A2夹紧位报警延时
LD 800.11  ; 夹爪A2夹紧位标志[0000.11]
AND 800.12  ; 夹爪A2松开位标志[0000.12]
ORLD
OR W400.11  ; [W400.11]夹爪A2夹紧位异常,请检查[0000.11]
ANDLD
ANDNOT 200.04  ; 报警清除
OUT W400.11  ; [W400.11]夹爪A2夹紧位异常,请检查[0000.11]
LD TR0
LD 10.12  ; 夹爪A2松开
ORNOT 800.11  ; 夹爪A2夹紧位标志[0000.11]
ANDLD
ANDNOT 800.12  ; 夹爪A2松开位标志[0000.12]
TIMX(550) 0112 D22  ; 报警长延时, 夹爪A2松开位报警延时
LD TR0
LD T0112  ; 夹爪A2松开位报警延时
LD 800.12  ; 夹爪A2松开位标志[0000.12]
AND 800.11  ; 夹爪A2夹紧位标志[0000.11]
ORLD
OR W400.12  ; [W400.12]夹爪A2松开位异常,请检查[0000.12]
ANDLD
ANDNOT 200.04  ; 报警清除
OUT W400.12  ; [W400.12]夹爪A2松开位异常,请检查[0000.12]

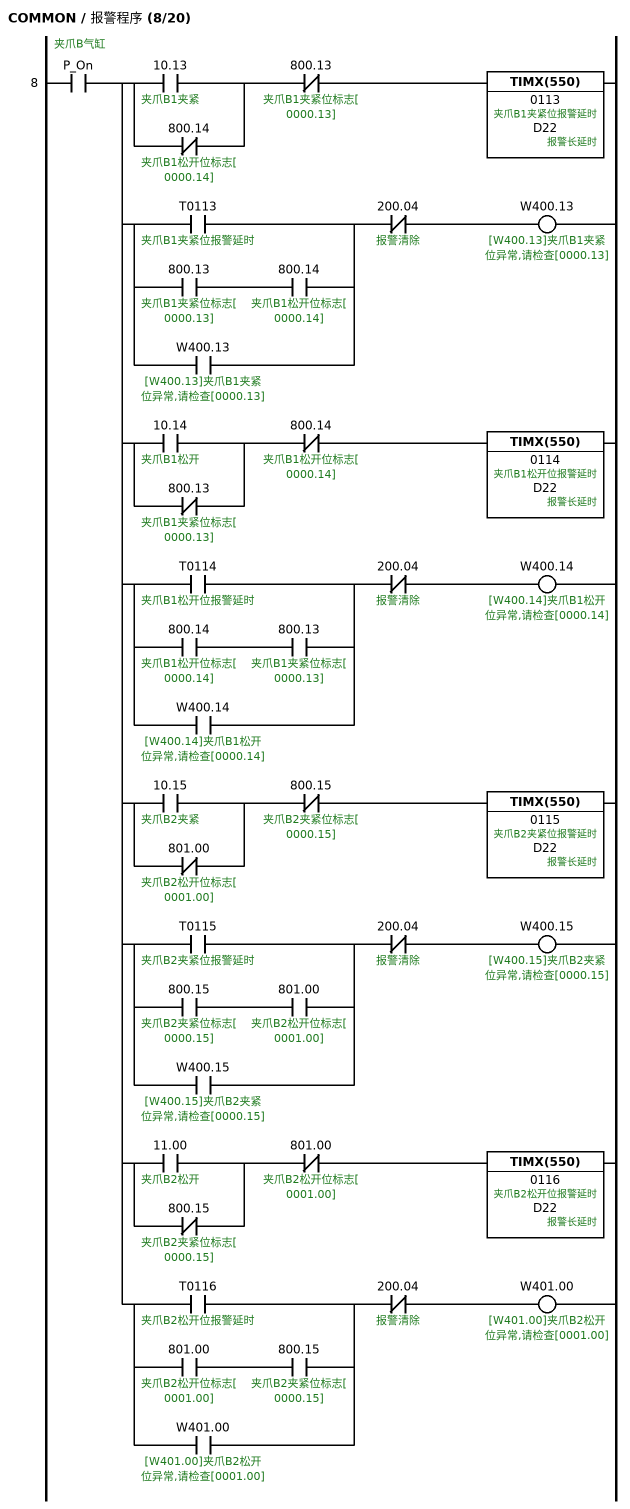
; rung 8: 夹爪B气缸
LD P_On
OUT TR0
LD 10.13  ; 夹爪B1夹紧
ORNOT 800.14  ; 夹爪B1松开位标志[0000.14]
ANDLD
ANDNOT 800.13  ; 夹爪B1夹紧位标志[0000.13]
TIMX(550) 0113 D22  ; 报警长延时, 夹爪B1夹紧位报警延时
LD TR0
LD T0113  ; 夹爪B1夹紧位报警延时
LD 800.13  ; 夹爪B1夹紧位标志[0000.13]
AND 800.14  ; 夹爪B1松开位标志[0000.14]
ORLD
OR W400.13  ; [W400.13]夹爪B1夹紧位异常,请检查[0000.13]
ANDLD
ANDNOT 200.04  ; 报警清除
OUT W400.13  ; [W400.13]夹爪B1夹紧位异常,请检查[0000.13]
LD TR0
LD 10.14  ; 夹爪B1松开
ORNOT 800.13  ; 夹爪B1夹紧位标志[0000.13]
ANDLD
ANDNOT 800.14  ; 夹爪B1松开位标志[0000.14]
TIMX(550) 0114 D22  ; 报警长延时, 夹爪B1松开位报警延时
LD TR0
LD T0114  ; 夹爪B1松开位报警延时
LD 800.14  ; 夹爪B1松开位标志[0000.14]
AND 800.13  ; 夹爪B1夹紧位标志[0000.13]
ORLD
OR W400.14  ; [W400.14]夹爪B1松开位异常,请检查[0000.14]
ANDLD
ANDNOT 200.04  ; 报警清除
OUT W400.14  ; [W400.14]夹爪B1松开位异常,请检查[0000.14]
LD TR0
LD 10.15  ; 夹爪B2夹紧
ORNOT 801.00  ; 夹爪B2松开位标志[0001.00]
ANDLD
ANDNOT 800.15  ; 夹爪B2夹紧位标志[0000.15]
TIMX(550) 0115 D22  ; 报警长延时, 夹爪B2夹紧位报警延时
LD TR0
LD T0115  ; 夹爪B2夹紧位报警延时
LD 800.15  ; 夹爪B2夹紧位标志[0000.15]
AND 801.00  ; 夹爪B2松开位标志[0001.00]
ORLD
OR W400.15  ; [W400.15]夹爪B2夹紧位异常,请检查[0000.15]
ANDLD
ANDNOT 200.04  ; 报警清除
OUT W400.15  ; [W400.15]夹爪B2夹紧位异常,请检查[0000.15]
LD TR0
LD 11.00  ; 夹爪B2松开
ORNOT 800.15  ; 夹爪B2夹紧位标志[0000.15]
ANDLD
ANDNOT 801.00  ; 夹爪B2松开位标志[0001.00]
TIMX(550) 0116 D22  ; 报警长延时, 夹爪B2松开位报警延时
LD TR0
LD T0116  ; 夹爪B2松开位报警延时
LD 801.00  ; 夹爪B2松开位标志[0001.00]
AND 800.15  ; 夹爪B2夹紧位标志[0000.15]
ORLD
OR W401.00  ; [W401.00]夹爪B2松开位异常,请检查[0001.00]
ANDLD
ANDNOT 200.04  ; 报警清除
OUT W401.00  ; [W401.00]夹爪B2松开位异常,请检查[0001.00]

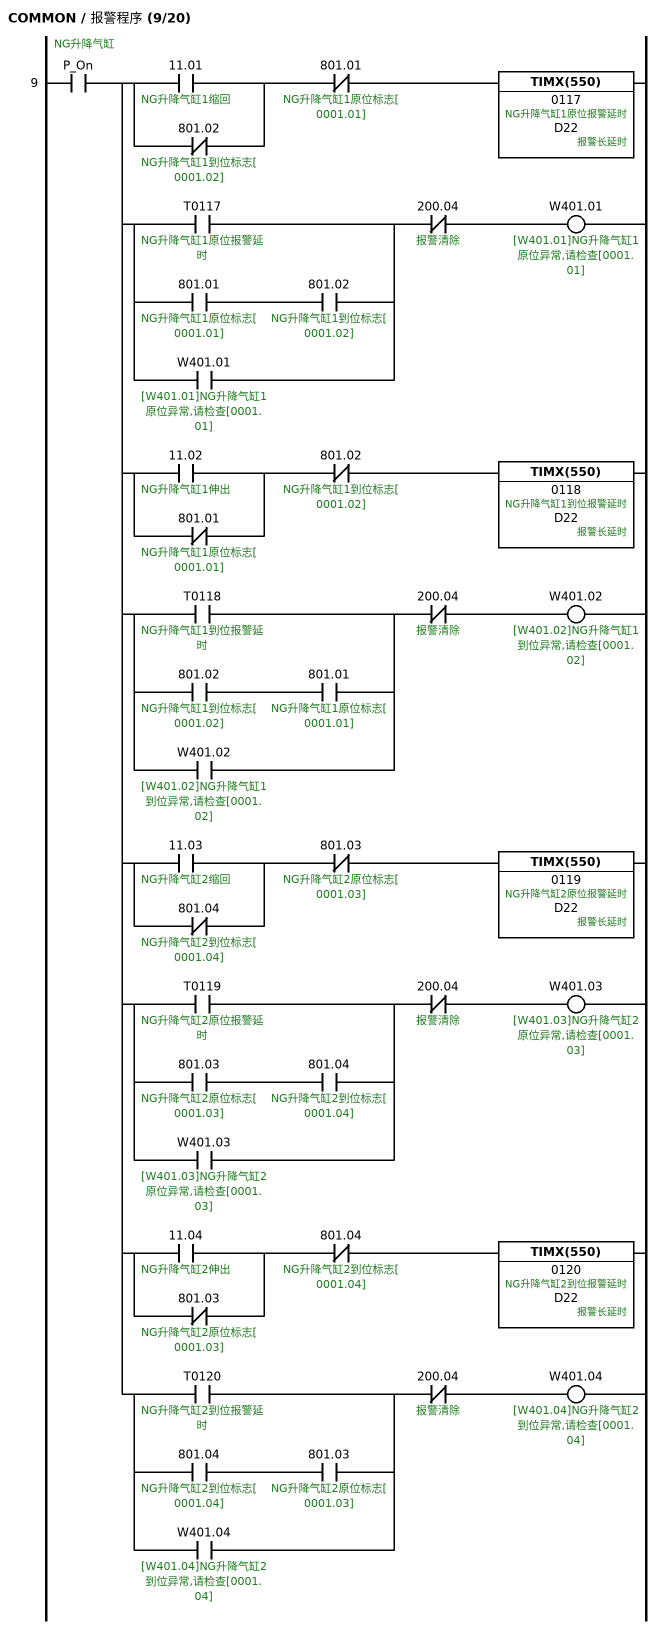
; rung 9: NG升降气缸
LD P_On
OUT TR0
LD 11.01  ; NG升降气缸1缩回
ORNOT 801.02  ; NG升降气缸1到位标志[0001.02]
ANDLD
ANDNOT 801.01  ; NG升降气缸1原位标志[0001.01]
TIMX(550) 0117 D22  ; 报警长延时, NG升降气缸1原位报警延时
LD TR0
LD T0117  ; NG升降气缸1原位报警延时
LD 801.01  ; NG升降气缸1原位标志[0001.01]
AND 801.02  ; NG升降气缸1到位标志[0001.02]
ORLD
OR W401.01  ; [W401.01]NG升降气缸1原位异常,请检查[0001.01]
ANDLD
ANDNOT 200.04  ; 报警清除
OUT W401.01  ; [W401.01]NG升降气缸1原位异常,请检查[0001.01]
LD TR0
LD 11.02  ; NG升降气缸1伸出
ORNOT 801.01  ; NG升降气缸1原位标志[0001.01]
ANDLD
ANDNOT 801.02  ; NG升降气缸1到位标志[0001.02]
TIMX(550) 0118 D22  ; 报警长延时, NG升降气缸1到位报警延时
LD TR0
LD T0118  ; NG升降气缸1到位报警延时
LD 801.02  ; NG升降气缸1到位标志[0001.02]
AND 801.01  ; NG升降气缸1原位标志[0001.01]
ORLD
OR W401.02  ; [W401.02]NG升降气缸1到位异常,请检查[0001.02]
ANDLD
ANDNOT 200.04  ; 报警清除
OUT W401.02  ; [W401.02]NG升降气缸1到位异常,请检查[0001.02]
LD TR0
LD 11.03  ; NG升降气缸2缩回
ORNOT 801.04  ; NG升降气缸2到位标志[0001.04]
ANDLD
ANDNOT 801.03  ; NG升降气缸2原位标志[0001.03]
TIMX(550) 0119 D22  ; 报警长延时, NG升降气缸2原位报警延时
LD TR0
LD T0119  ; NG升降气缸2原位报警延时
LD 801.03  ; NG升降气缸2原位标志[0001.03]
AND 801.04  ; NG升降气缸2到位标志[0001.04]
ORLD
OR W401.03  ; [W401.03]NG升降气缸2原位异常,请检查[0001.03]
ANDLD
ANDNOT 200.04  ; 报警清除
OUT W401.03  ; [W401.03]NG升降气缸2原位异常,请检查[0001.03]
LD TR0
LD 11.04  ; NG升降气缸2伸出
ORNOT 801.03  ; NG升降气缸2原位标志[0001.03]
ANDLD
ANDNOT 801.04  ; NG升降气缸2到位标志[0001.04]
TIMX(550) 0120 D22  ; 报警长延时, NG升降气缸2到位报警延时
LD TR0
LD T0120  ; NG升降气缸2到位报警延时
LD 801.04  ; NG升降气缸2到位标志[0001.04]
AND 801.03  ; NG升降气缸2原位标志[0001.03]
ORLD
OR W401.04  ; [W401.04]NG升降气缸2到位异常,请检查[0001.04]
ANDLD
ANDNOT 200.04  ; 报警清除
OUT W401.04  ; [W401.04]NG升降气缸2到位异常,请检查[0001.04]

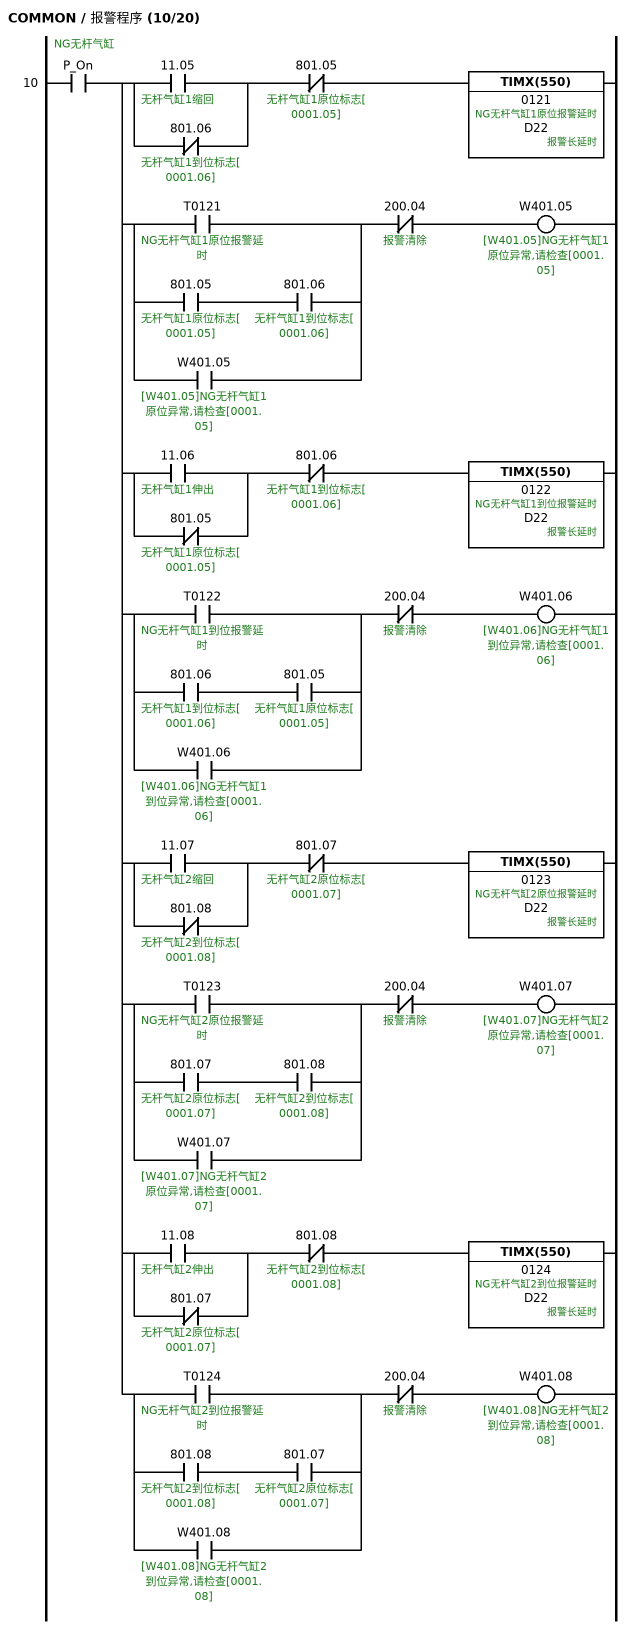
; rung 10: NG无杆气缸
LD P_On
OUT TR0
LD 11.05  ; 无杆气缸1缩回
ORNOT 801.06  ; 无杆气缸1到位标志[0001.06]
ANDLD
ANDNOT 801.05  ; 无杆气缸1原位标志[0001.05]
TIMX(550) 0121 D22  ; 报警长延时, NG无杆气缸1原位报警延时
LD TR0
LD T0121  ; NG无杆气缸1原位报警延时
LD 801.05  ; 无杆气缸1原位标志[0001.05]
AND 801.06  ; 无杆气缸1到位标志[0001.06]
ORLD
OR W401.05  ; [W401.05]NG无杆气缸1原位异常,请检查[0001.05]
ANDLD
ANDNOT 200.04  ; 报警清除
OUT W401.05  ; [W401.05]NG无杆气缸1原位异常,请检查[0001.05]
LD TR0
LD 11.06  ; 无杆气缸1伸出
ORNOT 801.05  ; 无杆气缸1原位标志[0001.05]
ANDLD
ANDNOT 801.06  ; 无杆气缸1到位标志[0001.06]
TIMX(550) 0122 D22  ; 报警长延时, NG无杆气缸1到位报警延时
LD TR0
LD T0122  ; NG无杆气缸1到位报警延时
LD 801.06  ; 无杆气缸1到位标志[0001.06]
AND 801.05  ; 无杆气缸1原位标志[0001.05]
ORLD
OR W401.06  ; [W401.06]NG无杆气缸1到位异常,请检查[0001.06]
ANDLD
ANDNOT 200.04  ; 报警清除
OUT W401.06  ; [W401.06]NG无杆气缸1到位异常,请检查[0001.06]
LD TR0
LD 11.07  ; 无杆气缸2缩回
ORNOT 801.08  ; 无杆气缸2到位标志[0001.08]
ANDLD
ANDNOT 801.07  ; 无杆气缸2原位标志[0001.07]
TIMX(550) 0123 D22  ; 报警长延时, NG无杆气缸2原位报警延时
LD TR0
LD T0123  ; NG无杆气缸2原位报警延时
LD 801.07  ; 无杆气缸2原位标志[0001.07]
AND 801.08  ; 无杆气缸2到位标志[0001.08]
ORLD
OR W401.07  ; [W401.07]NG无杆气缸2原位异常,请检查[0001.07]
ANDLD
ANDNOT 200.04  ; 报警清除
OUT W401.07  ; [W401.07]NG无杆气缸2原位异常,请检查[0001.07]
LD TR0
LD 11.08  ; 无杆气缸2伸出
ORNOT 801.07  ; 无杆气缸2原位标志[0001.07]
ANDLD
ANDNOT 801.08  ; 无杆气缸2到位标志[0001.08]
TIMX(550) 0124 D22  ; 报警长延时, NG无杆气缸2到位报警延时
LD TR0
LD T0124  ; NG无杆气缸2到位报警延时
LD 801.08  ; 无杆气缸2到位标志[0001.08]
AND 801.07  ; 无杆气缸2原位标志[0001.07]
ORLD
OR W401.08  ; [W401.08]NG无杆气缸2到位异常,请检查[0001.08]
ANDLD
ANDNOT 200.04  ; 报警清除
OUT W401.08  ; [W401.08]NG无杆气缸2到位异常,请检查[0001.08]

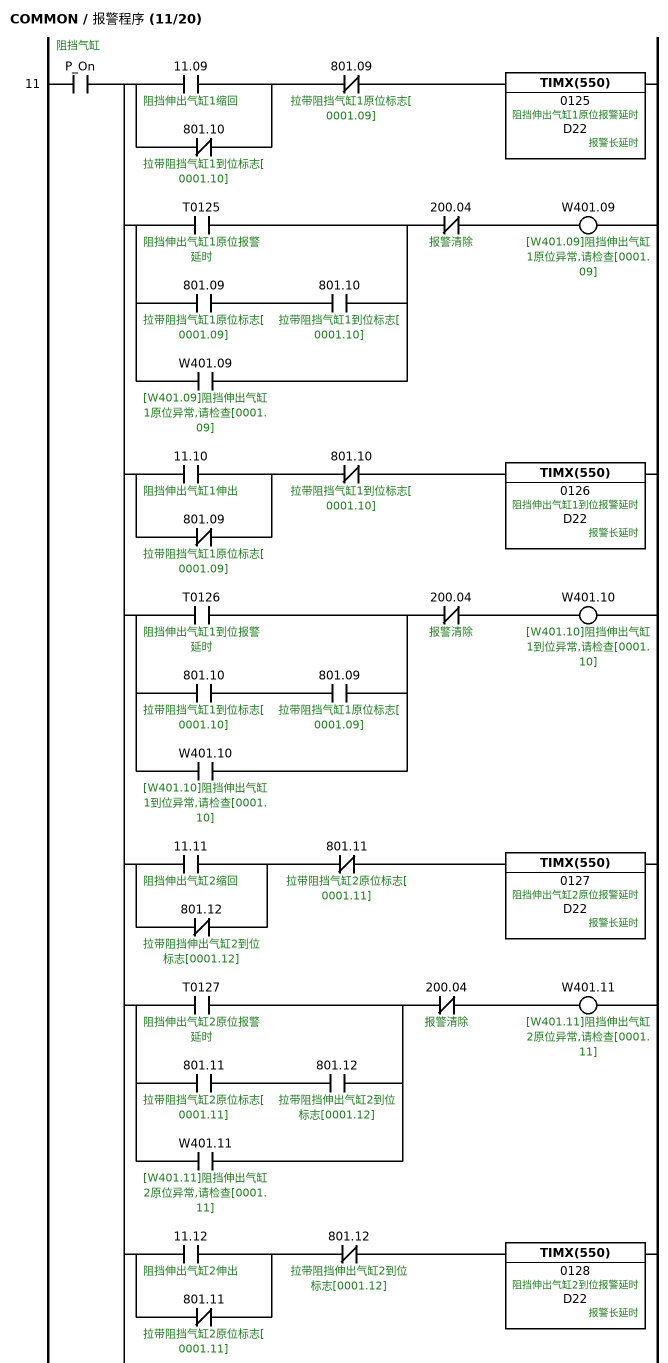

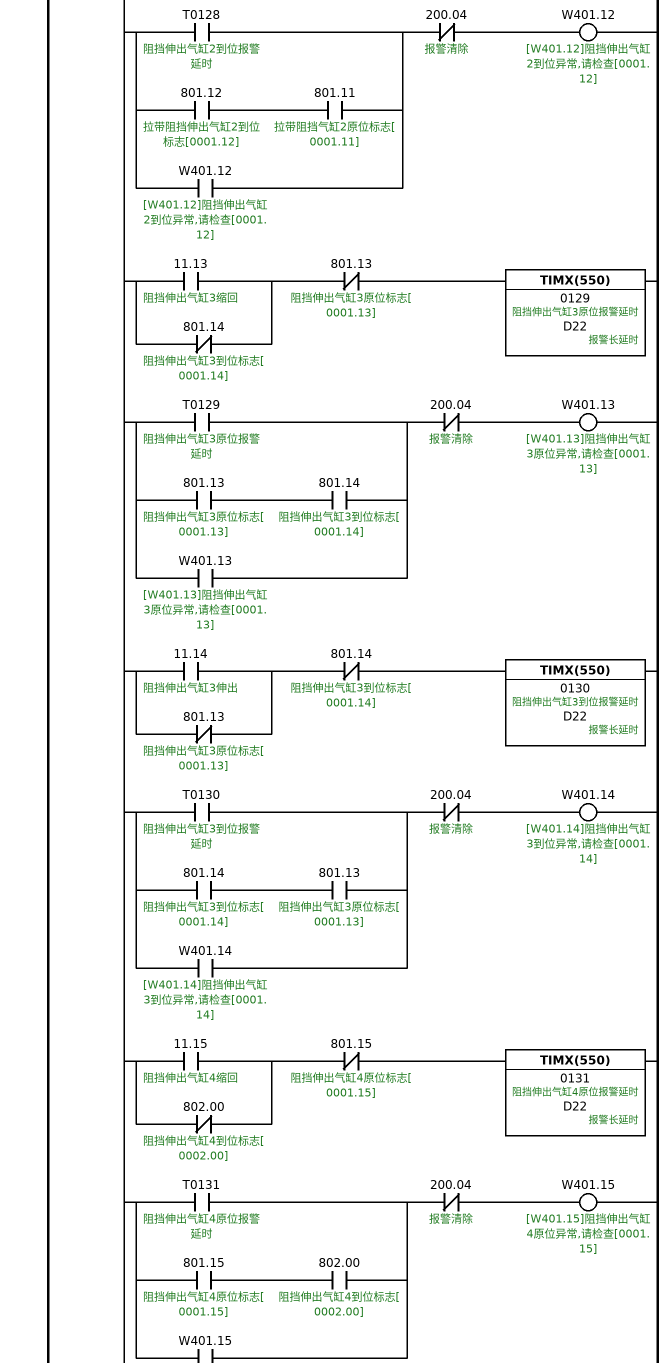

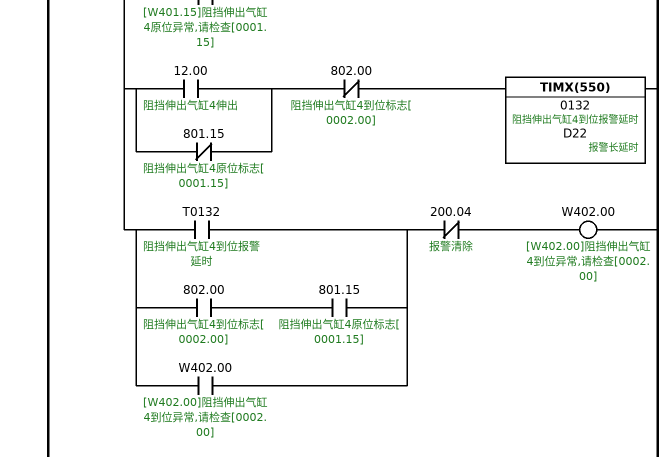
; rung 11: 阻挡气缸
LD P_On
OUT TR0
LD 11.09  ; 阻挡伸出气缸1缩回
ORNOT 801.10  ; 拉带阻挡气缸1到位标志[0001.10]
ANDLD
ANDNOT 801.09  ; 拉带阻挡气缸1原位标志[0001.09]
TIMX(550) 0125 D22  ; 报警长延时, 阻挡伸出气缸1原位报警延时
LD TR0
LD T0125  ; 阻挡伸出气缸1原位报警延时
LD 801.09  ; 拉带阻挡气缸1原位标志[0001.09]
AND 801.10  ; 拉带阻挡气缸1到位标志[0001.10]
ORLD
OR W401.09  ; [W401.09]阻挡伸出气缸1原位异常,请检查[0001.09]
ANDLD
ANDNOT 200.04  ; 报警清除
OUT W401.09  ; [W401.09]阻挡伸出气缸1原位异常,请检查[0001.09]
LD TR0
LD 11.10  ; 阻挡伸出气缸1伸出
ORNOT 801.09  ; 拉带阻挡气缸1原位标志[0001.09]
ANDLD
ANDNOT 801.10  ; 拉带阻挡气缸1到位标志[0001.10]
TIMX(550) 0126 D22  ; 报警长延时, 阻挡伸出气缸1到位报警延时
LD TR0
LD T0126  ; 阻挡伸出气缸1到位报警延时
LD 801.10  ; 拉带阻挡气缸1到位标志[0001.10]
AND 801.09  ; 拉带阻挡气缸1原位标志[0001.09]
ORLD
OR W401.10  ; [W401.10]阻挡伸出气缸1到位异常,请检查[0001.10]
ANDLD
ANDNOT 200.04  ; 报警清除
OUT W401.10  ; [W401.10]阻挡伸出气缸1到位异常,请检查[0001.10]
LD TR0
LD 11.11  ; 阻挡伸出气缸2缩回
ORNOT 801.12  ; 拉带阻挡伸出气缸2到位标志[0001.12]
ANDLD
ANDNOT 801.11  ; 拉带阻挡气缸2原位标志[0001.11]
TIMX(550) 0127 D22  ; 报警长延时, 阻挡伸出气缸2原位报警延时
LD TR0
LD T0127  ; 阻挡伸出气缸2原位报警延时
LD 801.11  ; 拉带阻挡气缸2原位标志[0001.11]
AND 801.12  ; 拉带阻挡伸出气缸2到位标志[0001.12]
ORLD
OR W401.11  ; [W401.11]阻挡伸出气缸2原位异常,请检查[0001.11]
ANDLD
ANDNOT 200.04  ; 报警清除
OUT W401.11  ; [W401.11]阻挡伸出气缸2原位异常,请检查[0001.11]
LD TR0
LD 11.12  ; 阻挡伸出气缸2伸出
ORNOT 801.11  ; 拉带阻挡气缸2原位标志[0001.11]
ANDLD
ANDNOT 801.12  ; 拉带阻挡伸出气缸2到位标志[0001.12]
TIMX(550) 0128 D22  ; 报警长延时, 阻挡伸出气缸2到位报警延时
LD TR0
LD T0128  ; 阻挡伸出气缸2到位报警延时
LD 801.12  ; 拉带阻挡伸出气缸2到位标志[0001.12]
AND 801.11  ; 拉带阻挡气缸2原位标志[0001.11]
ORLD
OR W401.12  ; [W401.12]阻挡伸出气缸2到位异常,请检查[0001.12]
ANDLD
ANDNOT 200.04  ; 报警清除
OUT W401.12  ; [W401.12]阻挡伸出气缸2到位异常,请检查[0001.12]
LD TR0
LD 11.13  ; 阻挡伸出气缸3缩回
ORNOT 801.14  ; 阻挡伸出气缸3到位标志[0001.14]
ANDLD
ANDNOT 801.13  ; 阻挡伸出气缸3原位标志[0001.13]
TIMX(550) 0129 D22  ; 报警长延时, 阻挡伸出气缸3原位报警延时
LD TR0
LD T0129  ; 阻挡伸出气缸3原位报警延时
LD 801.13  ; 阻挡伸出气缸3原位标志[0001.13]
AND 801.14  ; 阻挡伸出气缸3到位标志[0001.14]
ORLD
OR W401.13  ; [W401.13]阻挡伸出气缸3原位异常,请检查[0001.13]
ANDLD
ANDNOT 200.04  ; 报警清除
OUT W401.13  ; [W401.13]阻挡伸出气缸3原位异常,请检查[0001.13]
LD TR0
LD 11.14  ; 阻挡伸出气缸3伸出
ORNOT 801.13  ; 阻挡伸出气缸3原位标志[0001.13]
ANDLD
ANDNOT 801.14  ; 阻挡伸出气缸3到位标志[0001.14]
TIMX(550) 0130 D22  ; 报警长延时, 阻挡伸出气缸3到位报警延时
LD TR0
LD T0130  ; 阻挡伸出气缸3到位报警延时
LD 801.14  ; 阻挡伸出气缸3到位标志[0001.14]
AND 801.13  ; 阻挡伸出气缸3原位标志[0001.13]
ORLD
OR W401.14  ; [W401.14]阻挡伸出气缸3到位异常,请检查[0001.14]
ANDLD
ANDNOT 200.04  ; 报警清除
OUT W401.14  ; [W401.14]阻挡伸出气缸3到位异常,请检查[0001.14]
LD TR0
LD 11.15  ; 阻挡伸出气缸4缩回
ORNOT 802.00  ; 阻挡伸出气缸4到位标志[0002.00]
ANDLD
ANDNOT 801.15  ; 阻挡伸出气缸4原位标志[0001.15]
TIMX(550) 0131 D22  ; 报警长延时, 阻挡伸出气缸4原位报警延时
LD TR0
LD T0131  ; 阻挡伸出气缸4原位报警延时
LD 801.15  ; 阻挡伸出气缸4原位标志[0001.15]
AND 802.00  ; 阻挡伸出气缸4到位标志[0002.00]
ORLD
OR W401.15  ; [W401.15]阻挡伸出气缸4原位异常,请检查[0001.15]
ANDLD
ANDNOT 200.04  ; 报警清除
OUT W401.15  ; [W401.15]阻挡伸出气缸4原位异常,请检查[0001.15]
LD TR0
LD 12.00  ; 阻挡伸出气缸4伸出
ORNOT 801.15  ; 阻挡伸出气缸4原位标志[0001.15]
ANDLD
ANDNOT 802.00  ; 阻挡伸出气缸4到位标志[0002.00]
TIMX(550) 0132 D22  ; 报警长延时, 阻挡伸出气缸4到位报警延时
LD TR0
LD T0132  ; 阻挡伸出气缸4到位报警延时
LD 802.00  ; 阻挡伸出气缸4到位标志[0002.00]
AND 801.15  ; 阻挡伸出气缸4原位标志[0001.15]
ORLD
OR W402.00  ; [W402.00]阻挡伸出气缸4到位异常,请检查[0002.00]
ANDLD
ANDNOT 200.04  ; 报警清除
OUT W402.00  ; [W402.00]阻挡伸出气缸4到位异常,请检查[0002.00]

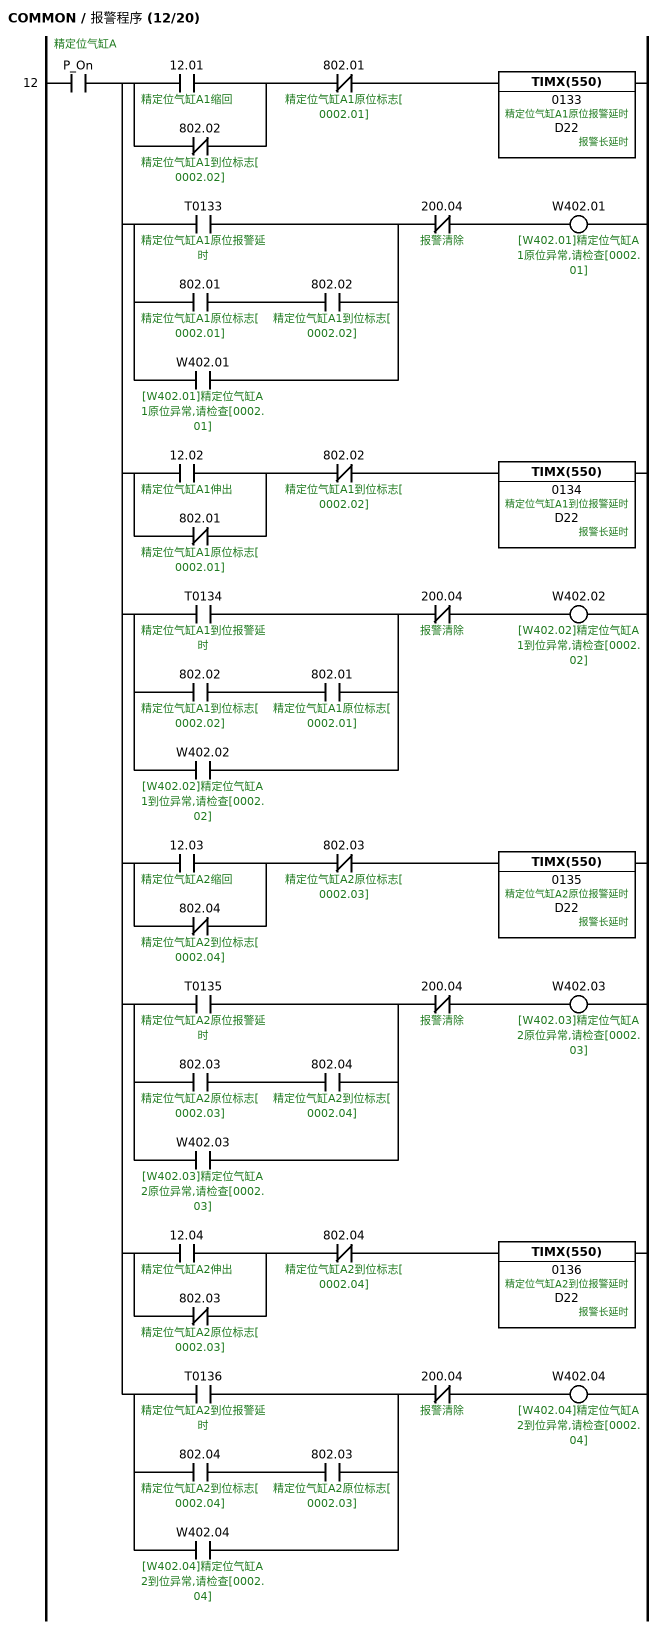
; rung 12: 精定位气缸A
LD P_On
OUT TR0
LD 12.01  ; 精定位气缸A1缩回
ORNOT 802.02  ; 精定位气缸A1到位标志[0002.02]
ANDLD
ANDNOT 802.01  ; 精定位气缸A1原位标志[0002.01]
TIMX(550) 0133 D22  ; 报警长延时, 精定位气缸A1原位报警延时
LD TR0
LD T0133  ; 精定位气缸A1原位报警延时
LD 802.01  ; 精定位气缸A1原位标志[0002.01]
AND 802.02  ; 精定位气缸A1到位标志[0002.02]
ORLD
OR W402.01  ; [W402.01]精定位气缸A1原位异常,请检查[0002.01]
ANDLD
ANDNOT 200.04  ; 报警清除
OUT W402.01  ; [W402.01]精定位气缸A1原位异常,请检查[0002.01]
LD TR0
LD 12.02  ; 精定位气缸A1伸出
ORNOT 802.01  ; 精定位气缸A1原位标志[0002.01]
ANDLD
ANDNOT 802.02  ; 精定位气缸A1到位标志[0002.02]
TIMX(550) 0134 D22  ; 报警长延时, 精定位气缸A1到位报警延时
LD TR0
LD T0134  ; 精定位气缸A1到位报警延时
LD 802.02  ; 精定位气缸A1到位标志[0002.02]
AND 802.01  ; 精定位气缸A1原位标志[0002.01]
ORLD
OR W402.02  ; [W402.02]精定位气缸A1到位异常,请检查[0002.02]
ANDLD
ANDNOT 200.04  ; 报警清除
OUT W402.02  ; [W402.02]精定位气缸A1到位异常,请检查[0002.02]
LD TR0
LD 12.03  ; 精定位气缸A2缩回
ORNOT 802.04  ; 精定位气缸A2到位标志[0002.04]
ANDLD
ANDNOT 802.03  ; 精定位气缸A2原位标志[0002.03]
TIMX(550) 0135 D22  ; 报警长延时, 精定位气缸A2原位报警延时
LD TR0
LD T0135  ; 精定位气缸A2原位报警延时
LD 802.03  ; 精定位气缸A2原位标志[0002.03]
AND 802.04  ; 精定位气缸A2到位标志[0002.04]
ORLD
OR W402.03  ; [W402.03]精定位气缸A2原位异常,请检查[0002.03]
ANDLD
ANDNOT 200.04  ; 报警清除
OUT W402.03  ; [W402.03]精定位气缸A2原位异常,请检查[0002.03]
LD TR0
LD 12.04  ; 精定位气缸A2伸出
ORNOT 802.03  ; 精定位气缸A2原位标志[0002.03]
ANDLD
ANDNOT 802.04  ; 精定位气缸A2到位标志[0002.04]
TIMX(550) 0136 D22  ; 报警长延时, 精定位气缸A2到位报警延时
LD TR0
LD T0136  ; 精定位气缸A2到位报警延时
LD 802.04  ; 精定位气缸A2到位标志[0002.04]
AND 802.03  ; 精定位气缸A2原位标志[0002.03]
ORLD
OR W402.04  ; [W402.04]精定位气缸A2到位异常,请检查[0002.04]
ANDLD
ANDNOT 200.04  ; 报警清除
OUT W402.04  ; [W402.04]精定位气缸A2到位异常,请检查[0002.04]

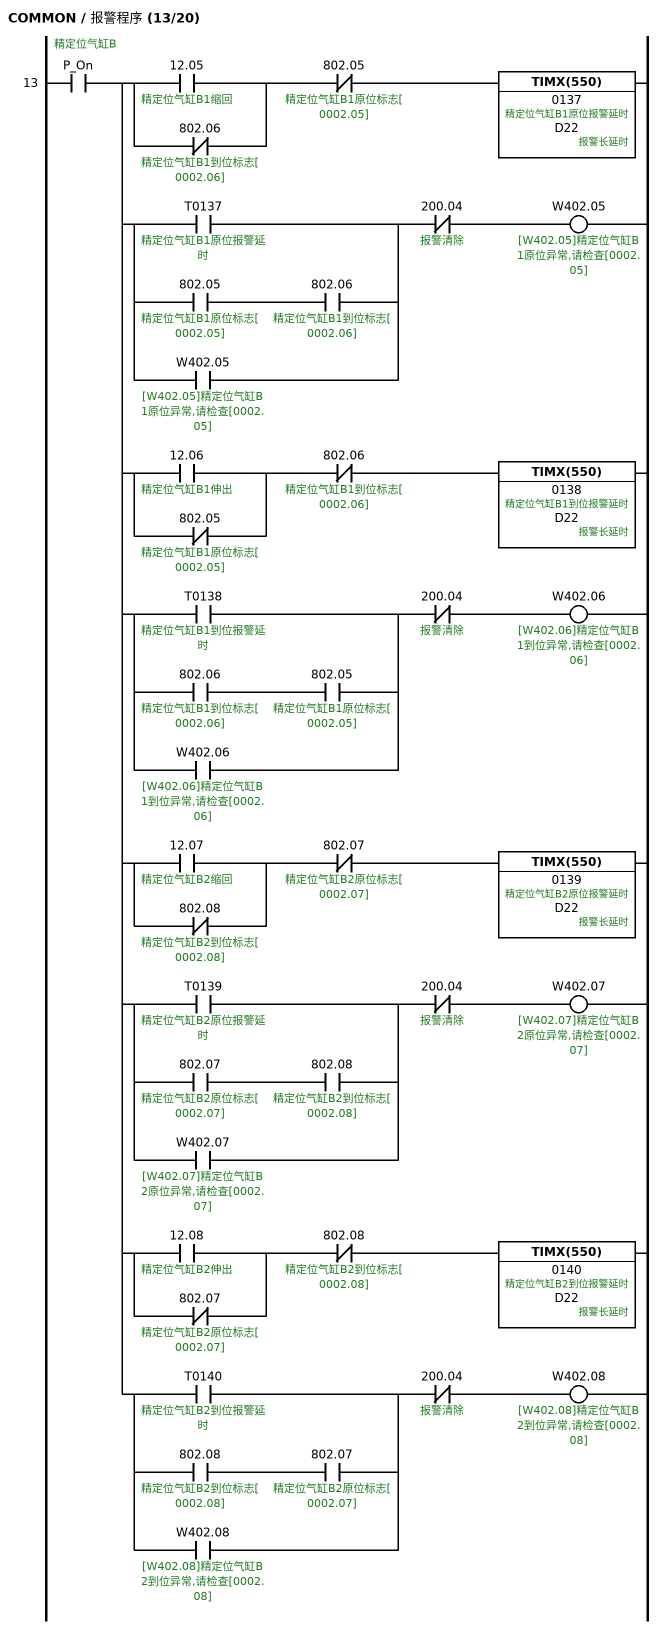
; rung 13: 精定位气缸B
LD P_On
OUT TR0
LD 12.05  ; 精定位气缸B1缩回
ORNOT 802.06  ; 精定位气缸B1到位标志[0002.06]
ANDLD
ANDNOT 802.05  ; 精定位气缸B1原位标志[0002.05]
TIMX(550) 0137 D22  ; 报警长延时, 精定位气缸B1原位报警延时
LD TR0
LD T0137  ; 精定位气缸B1原位报警延时
LD 802.05  ; 精定位气缸B1原位标志[0002.05]
AND 802.06  ; 精定位气缸B1到位标志[0002.06]
ORLD
OR W402.05  ; [W402.05]精定位气缸B1原位异常,请检查[0002.05]
ANDLD
ANDNOT 200.04  ; 报警清除
OUT W402.05  ; [W402.05]精定位气缸B1原位异常,请检查[0002.05]
LD TR0
LD 12.06  ; 精定位气缸B1伸出
ORNOT 802.05  ; 精定位气缸B1原位标志[0002.05]
ANDLD
ANDNOT 802.06  ; 精定位气缸B1到位标志[0002.06]
TIMX(550) 0138 D22  ; 报警长延时, 精定位气缸B1到位报警延时
LD TR0
LD T0138  ; 精定位气缸B1到位报警延时
LD 802.06  ; 精定位气缸B1到位标志[0002.06]
AND 802.05  ; 精定位气缸B1原位标志[0002.05]
ORLD
OR W402.06  ; [W402.06]精定位气缸B1到位异常,请检查[0002.06]
ANDLD
ANDNOT 200.04  ; 报警清除
OUT W402.06  ; [W402.06]精定位气缸B1到位异常,请检查[0002.06]
LD TR0
LD 12.07  ; 精定位气缸B2缩回
ORNOT 802.08  ; 精定位气缸B2到位标志[0002.08]
ANDLD
ANDNOT 802.07  ; 精定位气缸B2原位标志[0002.07]
TIMX(550) 0139 D22  ; 报警长延时, 精定位气缸B2原位报警延时
LD TR0
LD T0139  ; 精定位气缸B2原位报警延时
LD 802.07  ; 精定位气缸B2原位标志[0002.07]
AND 802.08  ; 精定位气缸B2到位标志[0002.08]
ORLD
OR W402.07  ; [W402.07]精定位气缸B2原位异常,请检查[0002.07]
ANDLD
ANDNOT 200.04  ; 报警清除
OUT W402.07  ; [W402.07]精定位气缸B2原位异常,请检查[0002.07]
LD TR0
LD 12.08  ; 精定位气缸B2伸出
ORNOT 802.07  ; 精定位气缸B2原位标志[0002.07]
ANDLD
ANDNOT 802.08  ; 精定位气缸B2到位标志[0002.08]
TIMX(550) 0140 D22  ; 报警长延时, 精定位气缸B2到位报警延时
LD TR0
LD T0140  ; 精定位气缸B2到位报警延时
LD 802.08  ; 精定位气缸B2到位标志[0002.08]
AND 802.07  ; 精定位气缸B2原位标志[0002.07]
ORLD
OR W402.08  ; [W402.08]精定位气缸B2到位异常,请检查[0002.08]
ANDLD
ANDNOT 200.04  ; 报警清除
OUT W402.08  ; [W402.08]精定位气缸B2到位异常,请检查[0002.08]

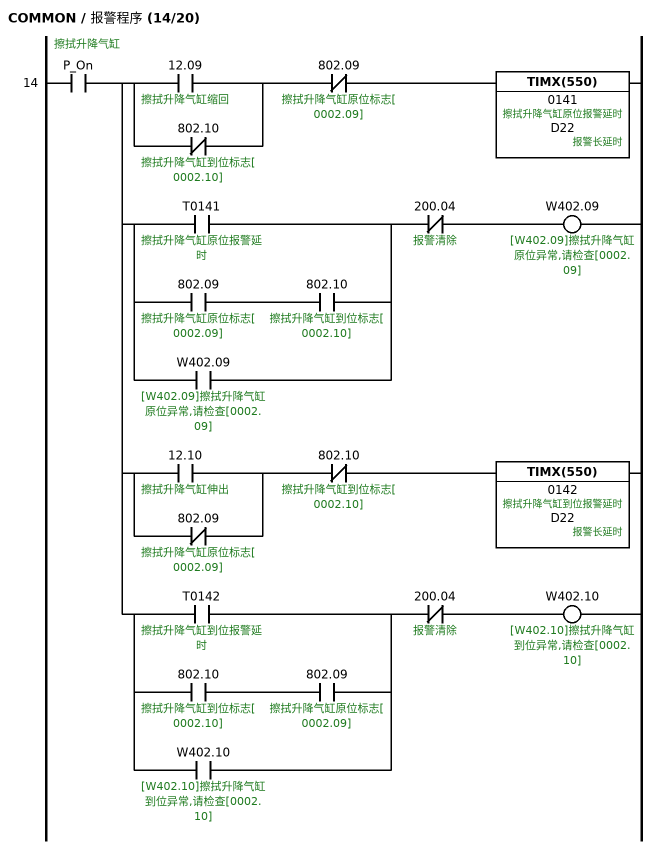
; rung 14: 擦拭升降气缸
LD P_On
OUT TR0
LD 12.09  ; 擦拭升降气缸缩回
ORNOT 802.10  ; 擦拭升降气缸到位标志[0002.10]
ANDLD
ANDNOT 802.09  ; 擦拭升降气缸原位标志[0002.09]
TIMX(550) 0141 D22  ; 报警长延时, 擦拭升降气缸原位报警延时
LD TR0
LD T0141  ; 擦拭升降气缸原位报警延时
LD 802.09  ; 擦拭升降气缸原位标志[0002.09]
AND 802.10  ; 擦拭升降气缸到位标志[0002.10]
ORLD
OR W402.09  ; [W402.09]擦拭升降气缸原位异常,请检查[0002.09]
ANDLD
ANDNOT 200.04  ; 报警清除
OUT W402.09  ; [W402.09]擦拭升降气缸原位异常,请检查[0002.09]
LD TR0
LD 12.10  ; 擦拭升降气缸伸出
ORNOT 802.09  ; 擦拭升降气缸原位标志[0002.09]
ANDLD
ANDNOT 802.10  ; 擦拭升降气缸到位标志[0002.10]
TIMX(550) 0142 D22  ; 报警长延时, 擦拭升降气缸到位报警延时
LD TR0
LD T0142  ; 擦拭升降气缸到位报警延时
LD 802.10  ; 擦拭升降气缸到位标志[0002.10]
AND 802.09  ; 擦拭升降气缸原位标志[0002.09]
ORLD
OR W402.10  ; [W402.10]擦拭升降气缸到位异常,请检查[0002.10]
ANDLD
ANDNOT 200.04  ; 报警清除
OUT W402.10  ; [W402.10]擦拭升降气缸到位异常,请检查[0002.10]

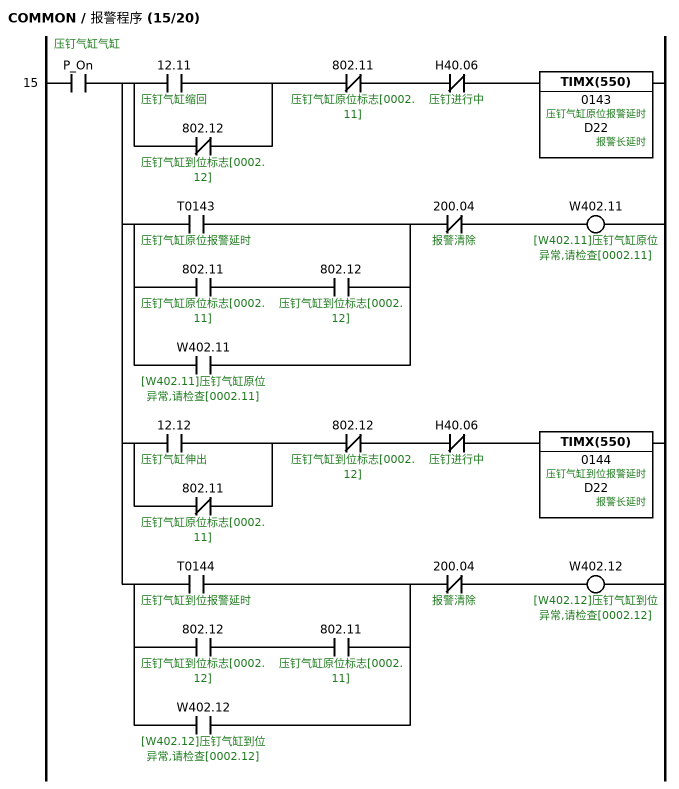
; rung 15: 压钉气缸气缸
LD P_On
OUT TR0
LD 12.11  ; 压钉气缸缩回
ORNOT 802.12  ; 压钉气缸到位标志[0002.12]
ANDLD
ANDNOT 802.11  ; 压钉气缸原位标志[0002.11]
ANDNOT H40.06  ; 压钉进行中
TIMX(550) 0143 D22  ; 报警长延时, 压钉气缸原位报警延时
LD TR0
LD T0143  ; 压钉气缸原位报警延时
LD 802.11  ; 压钉气缸原位标志[0002.11]
AND 802.12  ; 压钉气缸到位标志[0002.12]
ORLD
OR W402.11  ; [W402.11]压钉气缸原位异常,请检查[0002.11]
ANDLD
ANDNOT 200.04  ; 报警清除
OUT W402.11  ; [W402.11]压钉气缸原位异常,请检查[0002.11]
LD TR0
LD 12.12  ; 压钉气缸伸出
ORNOT 802.11  ; 压钉气缸原位标志[0002.11]
ANDLD
ANDNOT 802.12  ; 压钉气缸到位标志[0002.12]
ANDNOT H40.06  ; 压钉进行中
TIMX(550) 0144 D22  ; 报警长延时, 压钉气缸到位报警延时
LD TR0
LD T0144  ; 压钉气缸到位报警延时
LD 802.12  ; 压钉气缸到位标志[0002.12]
AND 802.11  ; 压钉气缸原位标志[0002.11]
ORLD
OR W402.12  ; [W402.12]压钉气缸到位异常,请检查[0002.12]
ANDLD
ANDNOT 200.04  ; 报警清除
OUT W402.12  ; [W402.12]压钉气缸到位异常,请检查[0002.12]

